rGoodStatistics[0]( CLK := stCycleDataNest1.LSS_Pass);
rBadStatistics[0]( CLK := stCycleDataNest1.LSS_Fail);
rGoodStatistics[1]( CLK := stCycleDataNest2.LSS_Pass);
rBadStatistics[1]( CLK := stCycleDataNest2.LSS_Fail);

IF 	rGoodStatistics[0].Q THEN
	
	stStatisticsHMI[4].nGood		:= stStatisticsHMI[4].nGood + 1;
	
END_IF
								
IF 	rBadStatistics[0].Q THEN
	
	stStatisticsHMI[4].nBad			:= stStatisticsHMI[4].nBad + 1;
	
END_IF

IF stStatisticsHMI[4].bResetGood THEN
	stStatisticsHMI[4].nGood		:= 0;
END_IF

IF stStatisticsHMI[4].bResetBad THEN
	stStatisticsHMI[4].nBad			:= 0;
END_IF

IF 	rGoodStatistics[1].Q THEN
	
	stStatisticsHMI[5].nGood		:= stStatisticsHMI[5].nGood + 1;
	
END_IF
								
IF 	rBadStatistics[1].Q THEN
	
	stStatisticsHMI[5].nBad			:= stStatisticsHMI[5].nBad + 1;
	
END_IF

IF stStatisticsHMI[5].bResetGood THEN
	stStatisticsHMI[5].nGood		:= 0;
END_IF

IF stStatisticsHMI[5].bResetBad THEN
	stStatisticsHMI[5].nBad			:= 0;
END_IF

IF (( stStatisticsHMI[4].nGood + stStatisticsHMI[4].nBad) <> 0) THEN
	
	rEfficency[0]							:= LREAL_TO_FMTSTR(in := (DINT_TO_REAL(stStatisticsHMI[4].nGood) /( DINT_TO_REAL(stStatisticsHMI[4].nGood) + DINT_TO_REAL(stStatisticsHMI[4].nBad))) * 100.0,iPrecision := 2, bRound := TRUE);
	stStatisticsHMI[4].nEfficency		:= CONCAT(STR1 := '%', STR2 := (rEfficency[0]));

ELSE stStatisticsHMI[4].nEfficency		:= CONCAT(STR1 := '%', STR2 := (DINT_TO_STRING(0)));
	
END_IF

IF (( stStatisticsHMI[5].nGood + stStatisticsHMI[5].nBad) <> 0) THEN
	
	rEfficency[1]							:= LREAL_TO_FMTSTR(in := (DINT_TO_REAL(stStatisticsHMI[5].nGood) /( DINT_TO_REAL(stStatisticsHMI[5].nGood) + DINT_TO_REAL(stStatisticsHMI[5].nBad))) * 100.0,iPrecision := 2, bRound := TRUE);
	stStatisticsHMI[5].nEfficency		:= CONCAT(STR1 := '%', STR2 := (rEfficency[1]));

ELSE stStatisticsHMI[5].nEfficency		:= CONCAT(STR1 := '%', STR2 := (DINT_TO_STRING(0)));
	
END_IF
END_ACTION

ACTION d_ACT_Set_Events_Station_3:
//IMMEDIATE FAULTS

stStationEvents[2].aEvents[0].bFault						:= TRUE;
stStationEvents[2].aEvents[0].bEventFlag					:= bError;
stStationEvents[2].aEvents[0].bEventText					:= 'Error Laser Snapshot';
stStationEvents[2].aEvents[0].sSolution						:= 'Check Laser Snapshot';


stStationEvents[2].aEvents[4].bFault						:= TRUE;
stStationEvents[2].aEvents[4].bEventTimer(IN := stLSS.Status.bBusy, PT := stTimers.tStation2TimeOut);
stStationEvents[2].aEvents[4].bEventFlag					:= stStationEvents[3].aEvents[4].bEventTimer.Q;
stStationEvents[2].aEvents[4].bEventText					:= 'Laser Snapshot Cycle Timeout';
stStationEvents[2].aEvents[4].sSolution						:= 'Reset Sytem';


//CYCLE STOP FAULT

stStationEvents[2].aEvents[24].bCycleStopRequest			:= TRUE;
stStationEvents[2].aEvents[24].bEventFlag					:= NOT bRun;
stStationEvents[2].aEvents[24].bEventText					:= 'Laser Snapshot is not in Run mode';
stStationEvents[2].aEvents[24].sSolution					:= 'Go to software and activate Run';
END_ACTION

ACTION e_ACT_HeightScalation:

//NEST LH
bScaledHeight1[1] := LSS_IO.nLH_HeightMeasurement_1-Offsets[1];
bScaledHeight1[2] := LSS_IO.nLH_HeightMeasurement_2-Offsets[2];
bScaledHeight1[3] := LSS_IO.nLH_HeightMeasurement_3-Offsets[3];
bScaledHeight1[4] := LSS_IO.nLH_HeightMeasurement_4-Offsets[4];
//NEST RH
bScaledHeight2[1] := LSS_IO.nRH_HeightMeasurement_1-Offsets[5];
bScaledHeight2[2] := LSS_IO.nRH_HeightMeasurement_2-Offsets[6];
bScaledHeight2[3] := LSS_IO.nRH_HeightMeasurement_3-Offsets[7];
bScaledHeight2[4] := LSS_IO.nRH_HeightMeasurement_4-Offsets[8];
END_ACTION

ACTION f_ACT_Measurement:

///////////////////////////////////////////////NEST 1//////////////////////////////////////////////
nHighLimit								:= nHeightSetPoint + nHeightTolerance;
nLowLimit								:= nHeightSetPoint - nHeightTolerance;
	

IF stLSS.CMD.LSS_CMD.Measurement1 THEN
	
IF 	(bScaledHeight1[1] < nHighLimit) AND
	(bScaledHeight1[1] > nLowLimit) THEN
									
	stCycleDataNest1.LSS_HeightPass[1]	:= TRUE;
	stCycleDataNest1.LSS_HeightFail[1]	:= FALSE;
									
ELSE
									
	stCycleDataNest1.LSS_HeightPass[1]	:= FALSE;
	stCycleDataNest1.LSS_HeightFail[1]	:= TRUE;
									
END_IF

IF 	(bScaledHeight1[2] < nHighLimit) AND
	(bScaledHeight1[2] > nLowLimit) THEN
									
	stCycleDataNest1.LSS_HeightPass[2]	:= TRUE;
	stCycleDataNest1.LSS_HeightFail[2]	:= FALSE;
									
ELSE
									
	stCycleDataNest1.LSS_HeightPass[2]	:= FALSE;
	stCycleDataNest1.LSS_HeightFail[2]	:= TRUE;
									
END_IF

IF 	(bScaledHeight1[3] < nHighLimit) AND
	(bScaledHeight1[3] > nLowLimit) THEN
									
	stCycleDataNest1.LSS_HeightPass[3]	:= TRUE;
	stCycleDataNest1.LSS_HeightFail[3]	:= FALSE;
									
ELSE
									
	stCycleDataNest1.LSS_HeightPass[3]	:= FALSE;
	stCycleDataNest1.LSS_HeightFail[3]	:= TRUE;
									
END_IF

IF 	(bScaledHeight1[4] < nHighLimit) AND
	(bScaledHeight1[4] > nLowLimit) THEN
									
	stCycleDataNest1.LSS_HeightPass[4]	:= TRUE;
	stCycleDataNest1.LSS_HeightFail[4]	:= FALSE;
									
ELSE
									
	stCycleDataNest1.LSS_HeightPass[4]	:= FALSE;
	stCycleDataNest1.LSS_HeightFail[4]	:= TRUE;
									
END_IF

IF stCycleDataNest1.LSS_HeightPass[1] AND stCycleDataNest1.LSS_HeightPass[2] AND
	stCycleDataNest1.LSS_HeightPass[3] AND stCycleDataNest1.LSS_HeightPass[4] THEN
	
	stCycleDataNest1.LSS_Pass			:= TRUE;
	stCycleDataNest1.LSS_Fail			:= FALSE;
	
ELSE 
	
	stCycleDataNest1.LSS_Pass			:= FALSE;
	stCycleDataNest1.LSS_Fail			:= TRUE;
	
END_IF

END_IF

///////////////////////////////////////////////NEST 2//////////////////////////////////////////////

IF stLSS.CMD.LSS_CMD.Measurement2 THEN
	
IF 	(bScaledHeight2[1] < nHighLimit) AND
	(bScaledHeight2[1] > nLowLimit) THEN
									
	stCycleDataNest2.LSS_HeightPass[1]	:= TRUE;
	stCycleDataNest2.LSS_HeightFail[1]	:= FALSE;
									
ELSE
									
	stCycleDataNest2.LSS_HeightPass[1]	:= FALSE;
	stCycleDataNest2.LSS_HeightFail[1]	:= TRUE;
									
END_IF

IF 	(bScaledHeight2[2] < nHighLimit) AND
	(bScaledHeight2[2] > nLowLimit) THEN
									
	stCycleDataNest2.LSS_HeightPass[2]	:= TRUE;
	stCycleDataNest2.LSS_HeightFail[2]	:= FALSE;
									
ELSE
									
	stCycleDataNest2.LSS_HeightPass[2]	:= FALSE;
	stCycleDataNest2.LSS_HeightFail[2]	:= TRUE;
									
END_IF

IF 	(bScaledHeight2[3] < nHighLimit) AND
	(bScaledHeight2[3] > nLowLimit) THEN
									
	stCycleDataNest2.LSS_HeightPass[3]	:= TRUE;
	stCycleDataNest2.LSS_HeightFail[3]	:= FALSE;
									
ELSE
									
	stCycleDataNest2.LSS_HeightPass[3]	:= FALSE;
	stCycleDataNest2.LSS_HeightFail[3]	:= TRUE;
									
END_IF

IF 	(bScaledHeight2[4] < nHighLimit) AND
	(bScaledHeight2[4] > nLowLimit) THEN
									
	stCycleDataNest2.LSS_HeightPass[4]	:= TRUE;
	stCycleDataNest2.LSS_HeightFail[4]	:= FALSE;
									
ELSE
									
	stCycleDataNest2.LSS_HeightPass[4]	:= FALSE;
	stCycleDataNest2.LSS_HeightFail[4]	:= TRUE;
									
END_IF

IF stCycleDataNest2.LSS_HeightPass[1] AND stCycleDataNest2.LSS_HeightPass[2] AND
	stCycleDataNest2.LSS_HeightPass[3] AND stCycleDataNest2.LSS_HeightPass[4] THEN
	
	stCycleDataNest2.LSS_Pass			:= TRUE;
	stCycleDataNest2.LSS_Fail			:= FALSE;
	
ELSE 
	
	stCycleDataNest2.LSS_Pass			:= FALSE;
	stCycleDataNest2.LSS_Fail			:= TRUE;
	
END_IF

END_IF
END_ACTION

ACTION g_ACT_Calibration:
tonCalibrationTrigger( IN := (bSetCalibrationHeight1 OR bSetCalibrationHeight2) AND (bResultsReady AND NOT bBusy), PT := T#500MS);

IF bSetCalibrationHeight1 THEN
	
	bTrigger										:= TRUE;
			
	CalibrationHeight1[1]						:= LSS_IO.nLH_HeightMeasurement_1;	
	CalibrationHeight1[2]						:= LSS_IO.nLH_HeightMeasurement_2;
	CalibrationHeight1[3]						:= LSS_IO.nLH_HeightMeasurement_3;
	CalibrationHeight1[4]						:= LSS_IO.nLH_HeightMeasurement_4;	

END_IF

IF bSetCalibrationHeight2 THEN
	
	bTrigger										:= TRUE;

	CalibrationHeight2[1]						:= LSS_IO.nRH_HeightMeasurement_1;	
	CalibrationHeight2[2]						:= LSS_IO.nRH_HeightMeasurement_2;
	CalibrationHeight2[3]						:= LSS_IO.nRH_HeightMeasurement_3;
	CalibrationHeight2[4]						:= LSS_IO.nRH_HeightMeasurement_4;

END_IF

IF tonCalibrationTrigger.Q THEN
	
	bSetCalibrationHeight1						:= FALSE;
	bSetCalibrationHeight2						:= FALSE;
	bResultsAcknowledge							:= TRUE;
	bTrigger									:= FALSE;
	

END_IF

tonResultAcknowledge(IN := NOT bSetCalibrationHeight1 AND NOT bSetCalibrationHeight2, PT := T#500MS);
rResultAcknowledge(CLK := tonResultAcknowledge.Q);

IF rResultAcknowledge.Q THEN
	
	bResultsAcknowledge							:= FALSE;

END_IF

Offsets[1]					:= CalibrationHeight1[1] - nHeightSetByCalibration;
Offsets[2]					:= CalibrationHeight1[2] - nHeightSetByCalibration;
Offsets[3]					:= CalibrationHeight1[3] - nHeightSetByCalibration;
Offsets[4]					:= CalibrationHeight1[4] - nHeightSetByCalibration;

Offsets[5]					:= CalibrationHeight2[1] - nHeightSetByCalibration;
Offsets[6]					:= CalibrationHeight2[2] - nHeightSetByCalibration;
Offsets[7]					:= CalibrationHeight2[3] - nHeightSetByCalibration;
Offsets[8]					:= CalibrationHeight2[4] - nHeightSetByCalibration;
END_ACTION

END_PROGRAM

// ---- POUs/B_STATIONS/B_3_CAMERA/B_3_1_PRG_Master_Camera.TcPOU
PROGRAM B_3_1_PRG_Master_Camera

VAR
	
	rGoodStatistics						: ARRAY [0..1] OF R_TRIG;
	rBadStatistics						: ARRAY [0..1] OF R_TRIG;
	rEfficency							: ARRAY [0..1] OF STRING(510);
	bEventsFlag							: ARRAY [0..100] OF BOOL;
/////////////////////////////////////////////////////////////////////////////////////I O/////////////////////////////////////////////////////////////////////////////////////	
	bError								: ARRAY [1..2] OF BOOL;
	rReset								: R_TRIG;
	bReset								: BOOL;
	bReady								: BOOL;
	bDone								: ARRAY [1..2] OF BOOL;
	bFail								: ARRAY [1..2] OF BOOL;
	bTrigger							: ARRAY [1..2] OF BOOL;
	bTriggerFail						: ARRAY [1..2] OF BOOL;
	bBusy								: ARRAY [1..2] OF BOOL;
	bGeneralBusy						: BOOL;
	bClearBuffer						: BOOL;
	tonTakingPicture					: TON;
	
	abReTakingPicture					: ARRAY [1..2] OF BOOL;

	
END_VAR

d_ACT_Set_Events_Station_3();
a_ACT_Ctrl_Station_3();
b_ACT_IO();
c_ACT_Statistics_Station_3();

ACTION a_ACT_Ctrl_Station_3:
/////////////////////////////////////////////////////////////////////////////////////UTILITIES/////////////////////////////////////////////////////////////////////////////////////
tonTakingPicture(IN := stCamera.State = E_Camera_State.TAKING_PICTURE_PART_PRESENT_INSPECTION OR
						stCamera.State = E_Camera_State.TAKING_PICTURE_CONTINUOUS_PART_PRESENT, PT := T#500MS);

/////////////////////////////////////////////////////////////////////////////////////CONDITIONS/////////////////////////////////////////////////////////////////////////////////////

IF bError[1] OR bError[2] OR stCamera.CMD.bAbort THEN
	
	stCamera.State						:= E_Camera_State.RESET_CMD;

END_IF

CASE stCamera.State OF
	
	E_Camera_State.ABORTED:
	
								
								
	
								IF  stCamera.CMD.bEnable THEN
									
									stCamera.State						:= E_Camera_State.HOMING;
								
								END_IF
													
	E_Camera_State.HOMING:
	
								IF bReady THEN
									
									stCamera.State						:= E_Camera_State.READY;
									
								END_IF
	
						
	E_Camera_State.READY:
								bClearBuffer							:= TRUE;
							
								IF stCamera.CMD.bExecute THEN
									
									IF stCamera.CMD.CameraCMD.PartPresent1 OR stCamera.CMD.CameraCMD.PartPresent2 THEN
										
										stCamera.State					:=	E_Camera_State.TAKING_PICTURE_PART_PRESENT_INSPECTION;
										
									ELSIF stCamera.CMD.CameraCMD.ContinuousPartPresent1 OR stCamera.CMD.CameraCMD.ContinuousPartPresent2 THEN
										
										stCamera.State					:=	E_Camera_State.TAKING_PICTURE_CONTINUOUS_PART_PRESENT;
										
									END_IF
									
								END_IF
	
	E_Camera_State.TAKING_PICTURE_PART_PRESENT_INSPECTION:
								
								bClearBuffer							:= FALSE;
								
								bTrigger[1]								:= stCamera.CMD.CameraCMD.PartPresent1;
								bTrigger[2]								:= stCamera.CMD.CameraCMD.PartPresent2;
								
								IF tonTakingPicture.Q THEN
									
									bTrigger[1]							:= FALSE;
									bTrigger[2]							:= FALSE;
								
									bPartPresentNest1 					:= Camera1_IO.bPartPresentResult;
									bPartPresentNest2 					:= Camera2_IO.bPartPresentResult;
								
									stCamera.State 						:= E_Camera_State.RESULTS;
																	
								END_IF
	
	E_Camera_State.TAKING_PICTURE_CONTINUOUS_PART_PRESENT:
	
								IF stPuls.bFlash2Hz THEN
									
									bTrigger[1] 						:= stCamera.CMD.CameraCMD.ContinuousPartPresent1;
									bTrigger[2] 						:= stCamera.CMD.CameraCMD.ContinuousPartPresent2;
									
								ELSE 
									
									bTrigger[1]							:= FALSE;
									bTrigger[2]							:= FALSE;
									
								END_IF
								
								IF tonTakingPicture.Q THEN
								
									bPartPresentNest1 					:= Camera1_IO.bPartPresentResult;
									bPartPresentNest2 					:= Camera2_IO.bPartPresentResult;
									
								END_IF
								
								IF NOT stCamera.CMD.CameraCMD.ContinuousPartPresent1 AND NOT stCamera.CMD.CameraCMD.ContinuousPartPresent2 THEN
									
									stCamera.State						:= E_Camera_State.RESET_CMD;
									
								END_IF

		E_Camera_State.RESULTS:		
			
								bTrigger[1]								:= FALSE;
								bTrigger[2]								:= FALSE;	
								
								IF (bPartPresentNest1 OR NOT stCamera.CMD.CameraCMD.PartPresent1) AND 
									(bPartPresentNest2 OR NOT stCamera.CMD.CameraCMD.PartPresent2) THEN
									
									stCycleDataNest1.Camera_Pass			:= Camera1_IO.bSeptumPositionResult;
									stCycleDataNest1.Camera_Fail			:= NOT Camera1_IO.bSeptumPositionResult;
									stCycleDataNest2.Camera_Pass			:= Camera2_IO.bSeptumPositionResult;
									stCycleDataNest2.Camera_Fail			:= NOT Camera2_IO.bSeptumPositionResult;
									
									
								END_IF
									
								
								stCamera.State							:= E_Camera_State.DONE;
								
		E_Camera_State.DONE:		
	
								IF stCamera.CMD.bAcknowledge THEN
									
									stCamera.CMD.bAcknowledge			:= FALSE;
									stCamera.State						:= E_Camera_State.RESET_CMD;
								
								END_IF
								
	E_Camera_State.RESET_CMD:						
	
								
									
								bTrigger[1]								:= FALSE;
								bTrigger[2]								:= FALSE;								
									
								IF  stCamera.CMD.bAbort THEN

									stCamera.State						:= E_Camera_State.ABORTED;
								
								ELSE 
									stCamera.State						:= E_Camera_State.READY;
								END_IF
									

ELSE stCamera.State						:= E_Camera_State.READY;
	
END_CASE
/////////////////////////////////////////////////////////////////////////////////////STATUS/////////////////////////////////////////////////////////////////////////////////////

stCamera.Status.bBusy		:= 	(stCamera.State	= E_Camera_State.TAKING_PICTURE_PART_PRESENT_INSPECTION) OR 
								(stCamera.State	= E_Camera_State.TAKING_PICTURE_CONTINUOUS_PART_PRESENT);
								
stCamera.Status.bDone		:=	stCamera.State	= E_Camera_State.DONE;
											
stCamera.Status.bError		:= 	stCamera.State	= E_Camera_State.ERROR;

stCamera.Status.bReady		:= 	stCamera.State	= E_Camera_State.READY;

stCamera.Status.bStopped	:= 	NOT stCamera.Status.bBusy;
END_ACTION

ACTION b_ACT_IO:


bError[1]								:= Camera1_IO.bError;
bError[2]								:= Camera2_IO.bError;

	
bReady									:=  (Camera1_IO.bReady AND Camera1_IO.bRun) AND (Camera2_IO.bReady AND Camera2_IO.bRun);
	
bDone[1]								:= Camera1_IO.bResultReady;
bDone[2]								:= Camera2_IO.bResultReady;
	
bGeneralBusy						:= bBusy[1] OR bBusy[2];



bBusy[1]								:= Camera1_IO.bBusy;
bBusy[2]								:= Camera2_IO.bBusy;

bTriggerFail[1]							:= Camera1_IO.bTriggerFail;
bTriggerFail[2]							:= Camera2_IO.bTriggerFail;

Camera1_IO.bReset						:= bReset;
Camera2_IO.bReset						:= bReset;

Camera1_IO.bTrigger						:= bTrigger[1] OR bCameraTrigger[1];	
Camera2_IO.bTrigger						:= bTrigger[2] OR bCameraTrigger[2];

IF bClearBuffer	THEN
	
	Camera1_IO.bClearBuffer				:= TRUE;
	Camera2_IO.bClearBuffer				:= TRUE;

ELSE

	Camera1_IO.bClearBuffer				:= FALSE;
	Camera2_IO.bClearBuffer				:= FALSE;

END_IF
	

//////////////////////////////////////////////////////////////////////HMI//////////////////////////////////////////////////////////////////////////////
bCameraSettingNo[1]						:= 2;
bCameraSettingNo[2]						:= 2;



Camera1_IO.bResetStatistics				:= bCameraResetStatistics[1];
Camera1_IO.bSettingNo					:= bCameraSettingNo[1];
Camera1_IO.bSettingVal					:= bCameraSettingVal[1];
Camera1_IO.bSetTreshold					:= bCameraSetTreshold[1];

Camera2_IO.bResetStatistics				:= bCameraResetStatistics[2];
Camera2_IO.bSettingNo					:= bCameraSettingNo[2];
Camera2_IO.bSettingVal					:= bCameraSettingVal[2];
Camera2_IO.bSetTreshold					:= bCameraSetTreshold[2];


//Camera1_IO.bTriggerFail

rReset( CLK := stCamera.CMD.bReset, Q => bReset);
END_ACTION

ACTION c_ACT_Statistics_Station_3:
stStatisticsHMI[6].sName			:= 'Vision System 1';
stStatisticsHMI[7].sName			:= 'Vision System 2';


rGoodStatistics[0]( CLK := stCycleDataNest1.Camera_Pass);
rBadStatistics[0]( CLK := stCycleDataNest1.Camera_Fail);
rGoodStatistics[1]( CLK := stCycleDataNest2.Camera_Pass);
rBadStatistics[1]( CLK := stCycleDataNest2.Camera_Fail);

IF 	rGoodStatistics[0].Q THEN
	
	stStatisticsHMI[6].nGood		:= stStatisticsHMI[6].nGood + 1;
	
END_IF
								
IF 	rBadStatistics[0].Q THEN
	
	stStatisticsHMI[6].nBad			:= stStatisticsHMI[6].nBad + 1;
	
END_IF

IF stStatisticsHMI[6].bResetGood THEN
	stStatisticsHMI[6].nGood		:= 0;
END_IF

IF stStatisticsHMI[6].bResetBad THEN
	stStatisticsHMI[6].nBad			:= 0;
END_IF

IF 	rGoodStatistics[1].Q THEN
	
	stStatisticsHMI[7].nGood		:= stStatisticsHMI[7].nGood + 1;
	
END_IF
								
IF 	rBadStatistics[1].Q THEN
	
	stStatisticsHMI[7].nBad			:= stStatisticsHMI[7].nBad + 1;
	
END_IF

IF stStatisticsHMI[7].bResetGood THEN
	stStatisticsHMI[7].nGood		:= 0;
END_IF

IF stStatisticsHMI[7].bResetBad THEN
	stStatisticsHMI[7].nBad			:= 0;
END_IF

IF (( stStatisticsHMI[6].nGood + stStatisticsHMI[6].nBad) <> 0) THEN
	
	rEfficency[0]							:= LREAL_TO_FMTSTR(in := (DINT_TO_REAL(stStatisticsHMI[6].nGood) /( DINT_TO_REAL(stStatisticsHMI[6].nGood) + DINT_TO_REAL(stStatisticsHMI[6].nBad))) * 100.0,iPrecision := 2, bRound := TRUE);
	stStatisticsHMI[6].nEfficency		:= CONCAT(STR1 := '%', STR2 := (rEfficency[0]));

ELSE stStatisticsHMI[6].nEfficency		:= CONCAT(STR1 := '%', STR2 := (DINT_TO_STRING(0)));
	
END_IF

IF (( stStatisticsHMI[7].nGood + stStatisticsHMI[7].nBad) <> 0) THEN
	
	rEfficency[1]							:= LREAL_TO_FMTSTR(in := (DINT_TO_REAL(stStatisticsHMI[7].nGood) /( DINT_TO_REAL(stStatisticsHMI[7].nGood) + DINT_TO_REAL(stStatisticsHMI[7].nBad))) * 100.0,iPrecision := 2, bRound := TRUE);
	stStatisticsHMI[7].nEfficency		:= CONCAT(STR1 := '%', STR2 := (rEfficency[1]));

ELSE stStatisticsHMI[7].nEfficency		:= CONCAT(STR1 := '%', STR2 := (DINT_TO_STRING(0)));
	
END_IF
END_ACTION

ACTION d_ACT_Set_Events_Station_3:
//IMMEDIATE FAULTS

stStationEvents[3].aEvents[0].bFault						:= TRUE;
stStationEvents[3].aEvents[0].bEventFlag					:= bError[1];
stStationEvents[3].aEvents[0].bEventText					:= 'Error camera 1';
stStationEvents[3].aEvents[0].sSolution						:= 'Check camera 1';

stStationEvents[3].aEvents[1].bFault						:= TRUE;
stStationEvents[3].aEvents[1].bEventFlag					:= bError[2];
stStationEvents[3].aEvents[1].bEventText					:= 'Error camera 2';
stStationEvents[3].aEvents[1].sSolution						:= 'Check camera 2';

stStationEvents[3].aEvents[4].bFault						:= TRUE;
stStationEvents[3].aEvents[4].bEventTimer(IN := stCamera.Status.bBusy, PT := stTimers.tStation3TimeOut);
stStationEvents[3].aEvents[4].bEventFlag					:= stStationEvents[3].aEvents[4].bEventTimer.Q;
stStationEvents[3].aEvents[4].bEventText					:= 'Camera Cycle Timeout';
stStationEvents[3].aEvents[4].sSolution						:= 'Reset Sytem';


//CYCLE STOP FAULT

stStationEvents[3].aEvents[20].bCycleStopRequest			:= TRUE;
stStationEvents[3].aEvents[20].bEventFlag					:= bTriggerFail[1];
stStationEvents[3].aEvents[20].bEventText					:= 'Trigger failed in camera 1';
stStationEvents[3].aEvents[20].sSolution					:= 'Check camera 1';

stStationEvents[3].aEvents[21].bCycleStopRequest			:= TRUE;
stStationEvents[3].aEvents[21].bEventFlag					:= bTriggerFail[2];
stStationEvents[3].aEvents[21].bEventText					:= 'Trigger failed in camera 2';
stStationEvents[3].aEvents[21].sSolution					:= 'Check camera 2';

stStationEvents[3].aEvents[24].bCycleStopRequest			:= TRUE;
stStationEvents[3].aEvents[24].bEventFlag					:= NOT Camera1_IO.bRun;
stStationEvents[3].aEvents[24].bEventText					:= 'Camera 1 is not in Run mode';
stStationEvents[3].aEvents[24].sSolution					:= 'Go to software and activate Run';

stStationEvents[3].aEvents[25].bCycleStopRequest			:= TRUE;
stStationEvents[3].aEvents[25].bEventFlag					:= NOT Camera2_IO.bRun;
stStationEvents[3].aEvents[25].bEventText					:= 'Camera 2 is not in Run mode';
stStationEvents[3].aEvents[25].sSolution					:= 'Go to software and activate Run';
END_ACTION

END_PROGRAM

// ---- POUs/B_STATIONS/B_1_LEAK_TEST/B_1_1_PRG_Master_Leak_Test.TcPOU
PROGRAM B_1_1_PRG_Master_Leak_Test

VAR

	tonStationStopped					: TON;
	tonExecute							: TON;
	rGoodStatistics						: ARRAY [0..1] OF R_TRIG;
	rBadStatistics						: ARRAY [0..1] OF R_TRIG;
	rEfficency							: ARRAY [0..1] OF STRING(510);
	
	tonWaitResults						: TON;
/////////////////////////////////////////////////////////////////////////////////////I O/////////////////////////////////////////////////////////////////////////////////////	

	bStopped							: ARRAY [0..1] OF BOOL;
	bError								: ARRAY [0..1] OF BOOL;
	bReady								: ARRAY [0..1] OF BOOL;
	bDone								: ARRAY [0..1] OF BOOL;
	bReset								: ARRAY [0..1] OF BOOL;
	bStart								: ARRAY [0..1] OF BOOL;
	bStop								: ARRAY [0..1] OF BOOL;	
	bBusy								: ARRAY [0..1] OF BOOL;	
	fLeakTestDone						: ARRAY [0..1] OF F_TRIG;	
	bLeakTestDone						: ARRAY [0..1] OF BOOL;	
	rPass								: ARRAY [0..1] OF R_TRIG;	
	bPass								: ARRAY [0..1] OF BOOL;	
	rFail								: ARRAY [0..1] OF R_TRIG;	
	bFail								: ARRAY [0..1] OF BOOL;
	rReset								: ARRAY [0..1] OF R_TRIG;

	
END_VAR

a_ACT_Ctrl_Station_1();
b_ACT_IO();
c_ACT_Statistics_Station_1();
d_ACT_Set_Events_Station_1();

ACTION a_ACT_Ctrl_Station_1:
/////////////////////////////////////////////////////////////////////////////////////UTILITIES/////////////////////////////////////////////////////////////////////////////////////
tonStationStopped( IN := bStopped[0] AND bStopped[1], PT := T#1S);
tonExecute(IN := stLeakTesters.State = E_LeakTester_State.RUN_LEAK_TESTERS, PT := T#500MS);
tonWaitResults(IN := (stLeakTesters.State = E_LeakTester_State.WAIT_RESULTS), PT := T#100MS);

/////////////////////////////////////////////////////////////////////////////////////CONDITIONS/////////////////////////////////////////////////////////////////////////////////////

IF stLeakTesters.CMD.bAbort OR bError[0] OR bError[1] THEN
								
	stLeakTesters.State											:= E_LeakTester_State.RESET;
	

END_IF



CASE stLeakTesters.State OF
	
	E_LeakTester_State.ABORTED:
	
								IF stLeakTesters.CMD.bEnable AND NOT bError[0] THEN
									stLeakTesters.State			:= E_LeakTester_State.HOMING;
								ELSIF bError[0] OR bError[1] THEN
									stLeakTesters.State			:= E_LeakTester_State.ERROR;
								END_IF
	
	E_LeakTester_State.HOMING:
	
								IF bReady[0] AND bReady[1] AND bStopped[0] AND bStopped[1] THEN
									stLeakTesters.State			:= E_LeakTester_State.READY;
								
								END_IF
								
	E_LeakTester_State.READY:
	
								IF stLeakTesters.CMD.bExecute THEN
									
									stLeakTesters.State			:= E_LeakTester_State.RUN_LEAK_TESTERS;
								
								END_IF
		
								
	E_LeakTester_State.RUN_LEAK_TESTERS:	
								
								IF stLeakTesters.CMD.LeakTestersCMD.RunLeakTester1 AND stLeakTesters.CMD.LeakTestersCMD.RunLeakTester2 THEN
										
										bStart[0]				:= TRUE;
										bStart[1]				:= TRUE;
									
								ELSIF stLeakTesters.CMD.LeakTestersCMD.RunLeakTester1 AND NOT stLeakTesters.CMD.LeakTestersCMD.RunLeakTester2 THEN
										
										bStart[0]				:= TRUE;
									
								ELSIF NOT stLeakTesters.CMD.LeakTestersCMD.RunLeakTester1 AND stLeakTesters.CMD.LeakTestersCMD.RunLeakTester2 THEN
										
										bStart[1]				:= TRUE;
									
								END_IF
								
								IF tonExecute.Q THEN
									
									stLeakTesters.State			:= E_LeakTester_State.WAIT_LEAK_TESTERS;
								
								END_IF
	
	E_LeakTester_State.WAIT_LEAK_TESTERS:
	
								IF stLeakTesters.CMD.LeakTestersCMD.RunLeakTester1 AND stLeakTesters.CMD.LeakTestersCMD.RunLeakTester2 THEN
										
										IF bLeakTestDone[0] AND bLeakTestDone[1] THEN
											
											stLeakTesters.State	:= E_LeakTester_State.WAIT_RESULTS;
											
										END_IF
									
								ELSIF stLeakTesters.CMD.LeakTestersCMD.RunLeakTester1 AND NOT stLeakTesters.CMD.LeakTestersCMD.RunLeakTester2 THEN
										
										IF bLeakTestDone[0]  THEN
											
											stLeakTesters.State	:= E_LeakTester_State.WAIT_RESULTS;
											
										END_IF
									
								ELSIF NOT stLeakTesters.CMD.LeakTestersCMD.RunLeakTester1 AND stLeakTesters.CMD.LeakTestersCMD.RunLeakTester2 THEN
										
										IF bLeakTestDone[1]  THEN
											
											stLeakTesters.State	:= E_LeakTester_State.WAIT_RESULTS;
											
										END_IF
									
								END_IF
	
	E_LeakTester_State.WAIT_RESULTS:
	
								IF tonWaitResults.Q THEN
									
									stLeakTesters.State	:= E_LeakTester_State.RESULTS;
									
								END_IF


		
	E_LeakTester_State.RESULTS:
								
								IF stLeakTesters.CMD.LeakTestersCMD.RunLeakTester1 THEN
									
									IF bPass[0] THEN
									
										stCycleDataNest1.LeakTest_Pass := TRUE;
										stCycleDataNest1.LeakTest_Fail := FALSE;
										
										stLeakTesters.State	:= E_LeakTester_State.DONE;
								
									ELSIF bFail[0] THEN
									
										stCycleDataNest1.LeakTest_Fail := TRUE;
										stCycleDataNest1.LeakTest_Pass := FALSE;
								
										stLeakTesters.State	:= E_LeakTester_State.DONE;
										
								END_IF
									
								END_IF
								
								IF stLeakTesters.CMD.LeakTestersCMD.RunLeakTester2 THEN
									
									IF bPass[1] THEN
									
										stCycleDataNest2.LeakTest_Pass := TRUE;
										stCycleDataNest2.LeakTest_Fail	:= FALSE;
										
										stLeakTesters.State	:= E_LeakTester_State.DONE;
								
									ELSIF bFail[1] THEN
									
										stCycleDataNest2.LeakTest_Fail	:= TRUE;
										stCycleDataNest2.LeakTest_Pass := FALSE;
										
										stLeakTesters.State	:= E_LeakTester_State.DONE;
								
								END_IF
									
								END_IF
								
								
								
		E_LeakTester_State.DONE:
								IF  stLeakTesters.CMD.bAcknowledge THEN
									
									stLeakTesters.CMD.bAcknowledge := FALSE;
									stLeakTesters.State			:= E_LeakTester_State.RESET;
									
								END_IF	
								
								
								
	E_LeakTester_State.RESET:
	

								bStart[0]						:= FALSE;
								bStart[1]						:= FALSE;
								bReset[0]						:= FALSE;
								bReset[1]						:= FALSE;
								bStop[0]						:= FALSE;
								bStop[1]						:= FALSE;
								bLeakTestDone[0]				:= FALSE;
								bLeakTestDone[1]				:= FALSE;
								bPass[0]						:= FALSE;
								bPass[1]						:= FALSE;
								bFail[0]						:= FALSE;
								bFail[1]						:= FALSE;
								
								IF bError[0] OR bError[1] THEN

									stLeakTesters.State		:= E_LeakTester_State.ERROR;

								ELSIF stLeakTesters.CMD.bAbort OR stLeakTesters.CMD.bEndCycle THEN
									
									stLeakTesters.State			:= E_LeakTester_State.ABORTED;
									
								ELSE stLeakTesters.State			:= E_LeakTester_State.READY;
								
								END_IF
								
								
								
	E_LeakTester_State.STOPPING: 
	
								bStop[0]						:= TRUE;
								bStop[1]						:= TRUE;
								
								IF tonStationStopped.Q THEN
									
									stLeakTesters.State			:= E_LeakTester_State.RESET;
									
								END_IF
	
	E_LeakTester_State.ERROR:
	
								IF NOT bError[0] AND bError[1] THEN
									
									stLeakTesters.State						:= E_LeakTester_State.ABORTED;
									
								END_IF

ELSE stLeakTesters.State := E_LeakTester_State.ABORTED;
	
END_CASE
/////////////////////////////////////////////////////////////////////////////////////STATUS/////////////////////////////////////////////////////////////////////////////////////

stLeakTesters.Status.bBusy	:= 	stLeakTesters.State = E_LeakTester_State.STOPPING OR
								stLeakTesters.State = E_LeakTester_State.HOMING OR
								stLeakTesters.State = E_LeakTester_State.RUN_LEAK_TESTERS OR
								stLeakTesters.State = E_LeakTester_State.WAIT_LEAK_TESTERS;

stLeakTesters.Status.bDone	:= 	stLeakTesters.State = E_LeakTester_State.DONE;

stLeakTesters.Status.bError	:= 	stLeakTesters.State = E_LeakTester_State.ERROR;	

stLeakTesters.Status.bReady	:=	stLeakTesters.State = E_LeakTester_State.READY;

stLeakTesters.Status.bStopped := NOT stLeakTesters.Status.bBusy;
END_ACTION

ACTION b_ACT_IO:


bStopped[0]								:= NOT LeakTester1_IO.sti28General_I_O.bTestActiveLiveData;
bStopped[1]								:= NOT LeakTester2_IO.sti28General_I_O.bTestActiveLiveData;
bError[0]								:= LeakTester1_IO.sti28General_I_O.bMalfunction;
bError[1]								:= LeakTester2_IO.sti28General_I_O.bMalfunction;
bReady[0]								:= LeakTester1_IO.sti28General_I_O.bInstrumentReady;
bReady[1]								:= LeakTester2_IO.sti28General_I_O.bInstrumentReady;
LeakTester1_IO.sti28General_I_O.bReset	:= bReset[0] OR bLeaktester1_Reset;	
LeakTester2_IO.sti28General_I_O.bReset	:= bReset[1] OR bLeaktester2_Reset;	
LeakTester1_IO.sti28General_I_O.bStart	:= bStart[0] OR bLeaktester1_Start;
LeakTester2_IO.sti28General_I_O.bStart	:= bStart[1] OR bLeaktester2_Start;
LeakTester1_IO.sti28General_I_O.bStop	:= bStop[0] OR bLeaktester1_Stop OR stLeakTesters.CMD.bAbort;
LeakTester2_IO.sti28General_I_O.bStop	:= bStop[1] OR bLeaktester2_Stop OR stLeakTesters.CMD.bAbort;



rReset[0](CLK := stLeakTesters.CMD.bReset, Q => bReset[0]);
rReset[1](CLK := stLeakTesters.CMD.bReset, Q => bReset[1]);

fLeakTestDone[0](CLK := LeakTester1_IO.sti28General_I_O.bTestActiveLiveData);
fLeakTestDone[1](CLK := LeakTester2_IO.sti28General_I_O.bTestActiveLiveData);
rPass[0](CLK := LeakTester1_IO.sti28General_I_O.bProgramAccept);
rPass[1](CLK := LeakTester2_IO.sti28General_I_O.bProgramAccept);
rFail[0](CLK := LeakTester1_IO.sti28General_I_O.bProgramReject);
rFail[1](CLK := LeakTester2_IO.sti28General_I_O.bProgramReject);



IF fLeakTestDone[0].Q THEN
	
	bLeakTestDone[0]					:= TRUE;
	
END_IF

IF fLeakTestDone[1].Q THEN
	
	bLeakTestDone[1]					:= TRUE;
	
END_IF

IF rPass[0].Q THEN
	
	bPass[0]							:= TRUE;

END_IF

IF rPass[1].Q THEN
	
	bPass[1]							:= TRUE;

END_IF

IF rFail[0].Q THEN
	
	bFail[0]							:= TRUE;

END_IF

IF rFail[1].Q THEN
	
	bFail[1]							:= TRUE;

END_IF
END_ACTION

ACTION c_ACT_Statistics_Station_1:
stStatisticsHMI[2].sName			:= 'LEAK TESTER 1';
stStatisticsHMI[3].sName			:= 'LEAK TESTER 2';


rGoodStatistics[0]( CLK := stCycleDataNest1.LeakTest_Pass );
rGoodStatistics[1]( CLK := stCycleDataNest2.LeakTest_Pass );
rBadStatistics[0] ( CLK := stCycleDataNest1.LeakTest_Fail );
rBadStatistics[1] ( CLK := stCycleDataNest2.LeakTest_Fail );

IF 	rGoodStatistics[0].Q THEN
	
	stStatisticsHMI[2].nGood		:= stStatisticsHMI[2].nGood + 1;
	
END_IF
								
IF 	rBadStatistics[0].Q THEN
	
	stStatisticsHMI[2].nBad			:= stStatisticsHMI[2].nBad + 1;
	
END_IF

IF stStatisticsHMI[2].bResetGood THEN
	stStatisticsHMI[2].nGood		:= 0;
END_IF

IF stStatisticsHMI[2].bResetBad THEN
	stStatisticsHMI[2].nBad			:= 0;
END_IF


IF 	rGoodStatistics[1].Q THEN
	
	stStatisticsHMI[3].nGood		:= stStatisticsHMI[3].nGood + 1;
	
END_IF
								
IF 	rBadStatistics[1].Q THEN
	
	stStatisticsHMI[3].nBad			:= stStatisticsHMI[3].nBad + 1;
	
END_IF

IF stStatisticsHMI[3].bResetGood THEN
	stStatisticsHMI[3].nGood		:= 0;
END_IF

IF stStatisticsHMI[3].bResetBad THEN
	stStatisticsHMI[3].nBad			:= 0;
END_IF



IF (( stStatisticsHMI[2].nGood + stStatisticsHMI[2].nBad) <> 0) THEN
	
	rEfficency[0]							:= LREAL_TO_FMTSTR(in := (DINT_TO_REAL(stStatisticsHMI[2].nGood) /( DINT_TO_REAL(stStatisticsHMI[2].nGood) + DINT_TO_REAL(stStatisticsHMI[2].nBad))) * 100.0,iPrecision := 2, bRound := TRUE);
	stStatisticsHMI[2].nEfficency		:= CONCAT(STR1 := '%', STR2 := (rEfficency[0]));

ELSE stStatisticsHMI[2].nEfficency		:= CONCAT(STR1 := '%', STR2 := (DINT_TO_STRING(0)));
	
END_IF

IF (( stStatisticsHMI[3].nGood + stStatisticsHMI[3].nBad) <> 0) THEN
	
	rEfficency[1]							:= LREAL_TO_FMTSTR(in := (DINT_TO_REAL(stStatisticsHMI[3].nGood) /( DINT_TO_REAL(stStatisticsHMI[3].nGood) + DINT_TO_REAL(stStatisticsHMI[3].nBad))) * 100.0,iPrecision := 2, bRound := TRUE);
	stStatisticsHMI[3].nEfficency		:= CONCAT(STR1 := '%', STR2 := (rEfficency[1]));

ELSE stStatisticsHMI[3].nEfficency		:= CONCAT(STR1 := '%', STR2 := (DINT_TO_STRING(0)));
	
END_IF
END_ACTION

ACTION d_ACT_Set_Events_Station_1:
//IMMEDIATE FAULTS

stStationEvents[1].aEvents[0].bFault						:= TRUE;
stStationEvents[1].aEvents[0].bEventTimer( IN := (stLeakTesters.State = E_LeakTester_State.RUN_LEAK_TESTERS) OR (stLeakTesters.State = E_LeakTester_State.WAIT_LEAK_TESTERS), PT := stTimers.tStation1TimeOut);
stStationEvents[1].aEvents[0].bEventFlag					:= stStationEvents[1].aEvents[0].bEventTimer.Q;
stStationEvents[1].aEvents[0].bEventText					:= 'Leak tester cycle Timeout';
stStationEvents[1].aEvents[0].sSolution						:= 'Reset System';



//CYCLE STOP REQUEST

stStationEvents[1].aEvents[20].bCycleStopRequest				:= TRUE;
stStationEvents[1].aEvents[20].bEventFlag					:= NOT bReady[0] AND (stLeakTesters.State = E_LeakTester_State.HOMING);// AND (stLeakTesters.State = E_LeakTester_State.HOMING);
stStationEvents[1].aEvents[20].bEventText					:= 'Leak Tester 1 not ready';
stStationEvents[1].aEvents[20].sSolution						:= 'Check Leak tester 1';

stStationEvents[1].aEvents[21].bCycleStopRequest				:= TRUE;
stStationEvents[1].aEvents[21].bEventFlag					:= NOT bReady[1] AND (stLeakTesters.State = E_LeakTester_State.HOMING);// AND (stLeakTesters.State = E_LeakTester_State.HOMING);
stStationEvents[1].aEvents[21].bEventText					:= 'Leak Tester 2 not ready';
stStationEvents[1].aEvents[21].sSolution						:= 'Check Leak tester 2';

stStationEvents[1].aEvents[22].bCycleStopRequest			:= TRUE;
stStationEvents[1].aEvents[22].bEventFlag					:= bError[0] AND bNest1Flag;
stStationEvents[1].aEvents[22].bEventText					:= 'Leak Tester 1 malfunction';
stStationEvents[1].aEvents[22].sSolution					:= 'Check Leak tester 1';

stStationEvents[1].aEvents[23].bCycleStopRequest			:= TRUE;
stStationEvents[1].aEvents[23].bEventFlag					:=  bError[1] AND bNest2Flag;
stStationEvents[1].aEvents[23].bEventText					:= 'Leak Tester 2 malfunction';
stStationEvents[1].aEvents[23].sSolution					:= 'Check Leak tester 2';

stStationEvents[1].aEvents[24].bCycleStopRequest			:= TRUE;
stStationEvents[1].aEvents[24].rEventTrigger( CLK := LeakTester1_IO.sti28LasResult.inPartEvaluation = 13);
stStationEvents[1].aEvents[24].bEventFlag					:=  stStationEvents[1].aEvents[24].rEventTrigger.Q;
stStationEvents[1].aEvents[24].bEventText					:= 'Leak Tester 1 Low Pressure';
stStationEvents[1].aEvents[24].sSolution					:= 'Check Leak tester 1 pneumatic circuit ';

stStationEvents[1].aEvents[25].bCycleStopRequest			:= TRUE;
stStationEvents[1].aEvents[25].rEventTrigger( CLK := LeakTester1_IO.sti28LasResult.inPartEvaluation = 14);
stStationEvents[1].aEvents[25].bEventFlag					:=  stStationEvents[1].aEvents[25].rEventTrigger.Q;
stStationEvents[1].aEvents[25].bEventText					:= 'Leak Tester 1 High Pressure';
stStationEvents[1].aEvents[25].sSolution					:= 'Check Leak tester 1 parameters';

stStationEvents[1].aEvents[26].bCycleStopRequest			:= TRUE;
stStationEvents[1].aEvents[26].rEventTrigger( CLK := LeakTester2_IO.sti28LasResult.inPartEvaluation = 13);
stStationEvents[1].aEvents[26].bEventFlag					:=  stStationEvents[1].aEvents[26].rEventTrigger.Q;
stStationEvents[1].aEvents[26].bEventText					:= 'Leak Tester 2 Low Pressure';
stStationEvents[1].aEvents[26].sSolution					:= 'Check Leak tester 2 pneumatic circuit ';

stStationEvents[1].aEvents[27].bCycleStopRequest			:= TRUE;
stStationEvents[1].aEvents[27].rEventTrigger( CLK := LeakTester2_IO.sti28LasResult.inPartEvaluation = 14);
stStationEvents[1].aEvents[27].bEventFlag					:=  stStationEvents[1].aEvents[27].rEventTrigger.Q;
stStationEvents[1].aEvents[27].bEventText					:= 'Leak Tester 2 High Pressure';
stStationEvents[1].aEvents[27].sSolution					:= 'Check Leak tester 2 parameters';

//Message
(*
stStationEvents[1].aEvents[3].bMessage						:= TRUE;
stStationEvents[1].aEvents[3].bEventFlag					:= bEventsFlag[3];
stStationEvents[1].aEvents[3].bEventText					:= 'Message 3';
stStationEvents[1].aEvents[3].sSolution						:= '';*)
END_ACTION

END_PROGRAM

// ---- POUs/B_STATIONS/B_4_PROCESS_CYLINDER__SLIDE_DOOR_VACUUM_CYLINDER/B_4_1_PRG_Master_ProcessCylinder.TcPOU
PROGRAM B_4_1_PRG_Master_ProcessCylinder

VAR

	
	
/////////////////////////////////////////////////////////////////////////////////////I O/////////////////////////////////////////////////////////////////////////////////////	
	bExtended							: ARRAY[1..2] OF BOOL;
	bRetracted							: ARRAY[1..2] OF BOOL;
	bExtend								: ARRAY[1..2] OF BOOL;
	bRetract							: ARRAY[1..2] OF BOOL;
	
	bHoldPart							: ARRAY[1..2] OF BOOL;
	tonPartReleased						: ARRAY[1..2] OF TON;
	tonHoldPart							: ARRAY[1..2] OF TON;
	
	bProcessDoorClosed					: BOOL;
	
END_VAR

d_ACT_Set_Events_Station_4A();
a_ACT_Ctrl_Station_4A();
b_ACT_IO_A();

ACTION a_ACT_Ctrl_Station_4A:
/////////////////////////////////////////////////////////////////////////////////////UTILITIES/////////////////////////////////////////////////////////////////////////////////////

IF stProcessCylinder.CMD.bAbort THEN
	
	stProcessCylinder.State												:= E_ProcessCylinder_State.RESET;
	bHoldPart[1]														:= FALSE;
	bHoldPart[2]														:= FALSE;

END_IF

/////////////////////////////////////////////////////////////////////////////////////CONDITIONS/////////////////////////////////////////////////////////////////////////////////////

CASE stProcessCylinder.State OF
	
	E_ProcessCylinder_State.ABORTED:
	
								IF stProcessCylinder.CMD.bEnable THEN
									
									stProcessCylinder.State				:= E_ProcessCylinder_State.HOMING;
								
								END_IF
								
	E_ProcessCylinder_State.HOMING:
	
								bHoldPart[1]							:= FALSE;
								bHoldPart[2]							:= FALSE;
	
								IF NOT bRetracted[1] AND (NOT bHoldPart[1] AND bProcessDoorClosed) THEN
									
									bRetract[1]							:= TRUE;
									
								END_IF
								
								IF NOT bRetracted[2] AND (NOT bHoldPart[2] AND bProcessDoorClosed) THEN
									
									bRetract[2]							:= TRUE;
									
								END_IF
								
								
								IF bRetracted[1] AND bRetracted[2] THEN
									
									bRetract[1]							:= FALSE;
									bRetract[2]							:= FALSE;
									stProcessCylinder.State				:= E_ProcessCylinder_State.READY;
									
								
								END_IF
	
	E_ProcessCylinder_State.READY:
	
								IF stProcessCylinder.CMD.bExecute AND (stProcessCylinder.CMD.ProcessCylinderCMD.ExtendCylinder1 OR stProcessCylinder.CMD.ProcessCylinderCMD.ExtendCylinder2) THEN

									stProcessCylinder.State				:= E_ProcessCylinder_State.EXTEND;
									
								ELSIF stProcessCylinder.CMD.bExecute AND (stProcessCylinder.CMD.ProcessCylinderCMD.RetractCylinder1 OR stProcessCylinder.CMD.ProcessCylinderCMD.RetractCylinder2) THEN
									
									stProcessCylinder.State				:= E_ProcessCylinder_State.RETRACT;

								ELSIF stProcessCylinder.CMD.bExecute AND (stProcessCylinder.CMD.ProcessCylinderCMD.ExtendPartHolder1 OR stProcessCylinder.CMD.ProcessCylinderCMD.ExtendPartHolder2) THEN

									stProcessCylinder.State				:= E_ProcessCylinder_State.HOLD_PART;	

								ELSIF stProcessCylinder.CMD.bExecute AND (stProcessCylinder.CMD.ProcessCylinderCMD.RetractPartHolder1 OR stProcessCylinder.CMD.ProcessCylinderCMD.RetractPartHolder2) THEN

									stProcessCylinder.State				:= E_ProcessCylinder_State.RELEASE_PART;			
																		
								END_IF
	
	E_ProcessCylinder_State.EXTEND:
	
								bExtend[1]									:= stProcessCylinder.CMD.ProcessCylinderCMD.ExtendCylinder1;
								bExtend[2]									:= stProcessCylinder.CMD.ProcessCylinderCMD.ExtendCylinder2;
								
								IF (bExtended[1] OR NOT stProcessCylinder.CMD.ProcessCylinderCMD.ExtendCylinder1) AND (bExtended[2] OR NOT stProcessCylinder.CMD.ProcessCylinderCMD.ExtendCylinder2) THEN
									
									stProcessCylinder.State			:= E_ProcessCylinder_State.DONE;

								END_IF
								
	E_ProcessCylinder_State.RETRACT:
	
								bRetract[1]									:= stProcessCylinder.CMD.ProcessCylinderCMD.RetractCylinder1;
								bRetract[2]									:= stProcessCylinder.CMD.ProcessCylinderCMD.RetractCylinder2;
								
								
								IF (bRetracted[1] OR NOT stProcessCylinder.CMD.ProcessCylinderCMD.RetractCylinder1) AND (bRetracted[2] OR NOT stProcessCylinder.CMD.ProcessCylinderCMD.RetractCylinder2) THEN
									
									stProcessCylinder.State			:= E_ProcessCylinder_State.DONE;

								END_IF
								
	E_ProcessCylinder_State.HOLD_PART:
	
								bHoldPart[1]								:= stProcessCylinder.CMD.ProcessCylinderCMD.ExtendPartHolder1;
								bHoldPart[2]								:= stProcessCylinder.CMD.ProcessCylinderCMD.ExtendPartHolder2;
								
								
								IF (tonHoldPart[1].Q OR NOT stProcessCylinder.CMD.ProcessCylinderCMD.ExtendPartHolder1) AND (tonHoldPart[2].Q OR NOT stProcessCylinder.CMD.ProcessCylinderCMD.ExtendPartHolder2) THEN
									
									stProcessCylinder.State			:= E_ProcessCylinder_State.DONE;

								END_IF
								
	E_ProcessCylinder_State.RELEASE_PART:
	
								bHoldPart[1]								:= FALSE;
								bHoldPart[2]								:= FALSE;
								
								
								IF (tonPartReleased[1].Q OR NOT stProcessCylinder.CMD.ProcessCylinderCMD.RetractPartHolder1) AND (tonPartReleased[2].Q OR NOT stProcessCylinder.CMD.ProcessCylinderCMD.RetractPartHolder2) THEN
									
									stProcessCylinder.State			:= E_ProcessCylinder_State.DONE;

								END_IF
								
	E_ProcessCylinder_State.DONE:
	
								IF stProcessCylinder.CMD.bAcknowledge THEN
									
									stProcessCylinder.CMD.bAcknowledge		:= FALSE;
									stProcessCylinder.State					:= E_ProcessCylinder_State.RESET;
								
								END_IF
	
	
	E_ProcessCylinder_State.RESET:	
	
								bExtend[1]									:= FALSE;								
								bRetract[1]									:= FALSE;
								bExtend[2]									:= FALSE;								
								bRetract[2]									:= FALSE;
								
								IF NOT stProcessCylinder.CMD.bAbort AND NOT stProcessCylinder.CMD.bEndCycle THEN
									
									stProcessCylinder.State					:= E_ProcessCylinder_State.READY;
									
								ELSE stProcessCylinder.State					:= E_ProcessCylinder_State.ABORTED;
								END_IF
									

ELSE stProcessCylinder.State	:= E_ProcessCylinder_State.ABORTED;
	
END_CASE
/////////////////////////////////////////////////////////////////////////////////////STATUS/////////////////////////////////////////////////////////////////////////////////////

stProcessCylinder.Status.bBusy		:= 	stProcessCylinder.State	= E_ProcessCylinder_State.EXTEND OR
										stProcessCylinder.State	= E_ProcessCylinder_State.RETRACT OR 
										stProcessCylinder.State	= E_ProcessCylinder_State.RELEASE_PART OR 
										stProcessCylinder.State	= E_ProcessCylinder_State.HOLD_PART OR 
										stProcessCylinder.State	= E_ProcessCylinder_State.STOPPING;
								
stProcessCylinder.Status.bDone		:=	stProcessCylinder.State	= E_ProcessCylinder_State.DONE;

stProcessCylinder.Status.bReady		:= 	stProcessCylinder.State	= E_ProcessCylinder_State.READY;

stProcessCylinder.Status.bStopped	:= 	NOT stProcessCylinder.Status.bBusy;

stProcessCylinder.Status.bHomed		:= bRetracted[1] AND bRetracted[2];
END_ACTION

ACTION b_ACT_IO_A:

bExtended[1]								:= dw_T08_EL1809.iProcessCylinderExtended1;
bRetracted[1]								:= dw_T08_EL1809.iProcessCylinderRetracted1;
bExtended[2]								:= dw_T08_EL1809.iProcessCylinderExtended2;
bRetracted[2]								:= dw_T08_EL1809.iProcessCylinderRetracted2;

IF (bHoldPart[1] OR bHoldPart1) AND bExtended[1] THEN
	
	dw_T09_EL2809.qPartHolder1				:= TRUE;
	
ELSE

 dw_T09_EL2809.qPartHolder1				:= FALSE;

END_IF

IF (bHoldPart[2] OR bHoldPart2) AND bExtended[2] THEN
	
	dw_T10_EL2809.qPartHolder2				:= TRUE;
	
ELSE dw_T10_EL2809.qPartHolder2				:= FALSE;

END_IF

tonHoldPart[1](IN := NOT dw_T09_EL2809.qPartHolder1, PT := T#1S);
tonHoldPart[2](IN := NOT dw_T10_EL2809.qPartHolder2, PT := T#1S);

tonPartReleased[1](IN := NOT bHoldPart[1], PT := T#1S);
tonPartReleased[2](IN := NOT bHoldPart[2], PT := T#1S);

IF (bExtend[1] OR bProcessCtlinderExtend1) AND (tonPartReleased[1].Q AND bProcessDoorClosed) THEN
	
	dw_T09_EL2809.qExtendProcessCylinder1	:= TRUE ;
	dw_T09_EL2809.qRetractProcessCylinder1	:= FALSE;

ELSIF (bRetract[1] OR bProcessCtlinderRetract1) AND (tonPartReleased[1].Q AND bProcessDoorClosed )  THEN
	
	dw_T09_EL2809.qExtendProcessCylinder1	:= FALSE;
	dw_T09_EL2809.qRetractProcessCylinder1	:= TRUE;
	
ELSIF stMachineStatus.bFault THEN
	
	dw_T09_EL2809.qExtendProcessCylinder1	:= FALSE;
	dw_T09_EL2809.qRetractProcessCylinder1	:= FALSE;

END_IF

IF (bExtend[2] OR bProcessCtlinderExtend2) AND (tonPartReleased[2].Q AND bProcessDoorClosed) THEN
	
	dw_T10_EL2809.qExtendProcessCylinder2	:= TRUE ;
	dw_T10_EL2809.qRetractProcessCylinder2	:= FALSE;

ELSIF (bRetract[2] OR bProcessCtlinderRetract2) AND (tonPartReleased[2].Q AND bProcessDoorClosed)  THEN
	
	dw_T10_EL2809.qExtendProcessCylinder2	:= FALSE;
	dw_T10_EL2809.qRetractProcessCylinder2	:= TRUE;
	
ELSIF stMachineStatus.bFault THEN
	
	dw_T10_EL2809.qExtendProcessCylinder2	:= FALSE;
	dw_T10_EL2809.qRetractProcessCylinder2	:= FALSE;

END_IF


bProcessDoorClosed := dw_T05_EL1918.iProcessDoorClosed1 AND dw_T05_EL1918.iProcessDoorClosed2 AND dw_T05_EL1918.iProcessDoorFB;


bEnable_Holder[1]							:= bExtended[1];
bEnable_Holder[2]							:= bExtended[2];

bEnable_ProcessCylinder[1]					:= bProcessDoorClosed AND tonHoldPart[1].Q;
bEnable_ProcessCylinder[2]					:= bProcessDoorClosed AND tonHoldPart[2].Q;

bPartHeld[1]								:= bExtended[1] AND dw_T09_EL2809.qPartHolder1;
bPartHeld[2]								:= bExtended[2] AND dw_T10_EL2809.qPartHolder2;
END_ACTION

ACTION d_ACT_Set_Events_Station_4A:
//FAULTS 0..9

stStationEvents[4].aEvents[0].bEventTimer( IN := (bExtend[1] AND NOT bExtended[1]), PT := T#3S);
stStationEvents[4].aEvents[0].bFault						:= TRUE;
stStationEvents[4].aEvents[0].bEventFlag					:= stStationEvents[3].aEvents[0].bEventTimer.Q;
stStationEvents[4].aEvents[0].bEventText					:= 'Process Cylinder 1 extend timeout';
stStationEvents[4].aEvents[0].sSolution						:= 'Check cylinder, neumatic connections and sensors';

stStationEvents[4].aEvents[1].bEventTimer( IN := (bRetract[1] AND NOT bRetracted[1]), PT := T#3S);
stStationEvents[4].aEvents[1].bFault						:= TRUE;
stStationEvents[4].aEvents[1].bEventFlag					:= stStationEvents[3].aEvents[1].bEventTimer.Q;
stStationEvents[4].aEvents[1].bEventText					:= 'Process Cylinder retract timeout';
stStationEvents[4].aEvents[1].sSolution						:= 'Check cylinder, neumatic connections and sensors';

stStationEvents[4].aEvents[2].bEventTimer( IN := (bExtend[2] AND NOT bExtended[2]), PT := T#3S);
stStationEvents[4].aEvents[2].bFault						:= TRUE;
stStationEvents[4].aEvents[2].bEventFlag					:= stStationEvents[3].aEvents[2].bEventTimer.Q;
stStationEvents[4].aEvents[2].bEventText					:= 'Process Cylinder 2 extend timeout';
stStationEvents[4].aEvents[2].sSolution						:= 'Check cylinder, neumatic connections and sensors';

stStationEvents[4].aEvents[2].bEventTimer( IN := (bRetract[2] AND NOT bRetracted[2]), PT := T#3S);
stStationEvents[4].aEvents[2].bFault						:= TRUE;
stStationEvents[4].aEvents[2].bEventFlag					:= stStationEvents[3].aEvents[3].bEventTimer.Q;
stStationEvents[4].aEvents[2].bEventText					:= 'Process Cylinder retract timeout';
stStationEvents[4].aEvents[2].sSolution						:= 'Check cylinder, neumatic connections and sensors';


//CYCLE STOP REQUEST 30..39

(*stStationEvents[3].aEvents[2].bCycleStopRequest			:= TRUE;
stStationEvents[3].aEvents[2].bEventFlag					:= ;
stStationEvents[3].aEvents[2].bEventText					:= 'ST1 EVENT 7';*)
END_ACTION

END_PROGRAM

// ---- POUs/B_STATIONS/B_4_PROCESS_CYLINDER__SLIDE_DOOR_VACUUM_CYLINDER/B_4_2_PRG_Master_ProcessDoor.TcPOU
PROGRAM B_4_2_PRG_Master_ProcessDoor

VAR

	bEventsFlag							: ARRAY [0..100] OF BOOL;
/////////////////////////////////////////////////////////////////////////////////////I O/////////////////////////////////////////////////////////////////////////////////////	
	
	bOpenDoor							: BOOL;
	bCloseDoor							: BOOL;
	bCloseDoorHMI						: BOOL;
	bOpenDoorHMI						: BOOL;
	bDoorClosed							: BOOL;
	tonDoorOpened						: TON;
	bDoorOpened							: BOOL;	
	
END_VAR

d_ACT_Set_Events_Station_4B();
a_ACT_Ctrl_Station_4B();
b_ACT_IO_B();
c_Manual();

ACTION a_ACT_Ctrl_Station_4B:
/////////////////////////////////////////////////////////////////////////////////////UTILITIES/////////////////////////////////////////////////////////////////////////////////////

/////////////////////////////////////////////////////////////////////////////////////CONDITIONS/////////////////////////////////////////////////////////////////////////////////////
IF stProcessDoor.State <> E_ProcessDoor_State.HOMING THEN
	
	bDoorClosingInitFlag											:= FALSE;

END_IF


IF stProcessDoor.CMD.bAbort THEN
	
	stProcessDoor.State				:= E_ProcessDoor_State.RESET;
	
ELSIF stProcessDoor.CMD.bEndCycle THEN
	
	stProcessDoor.State				:= E_ProcessDoor_State.STOPPING;

END_IF

CASE stProcessDoor.State OF
	
	E_ProcessDoor_State.ABORTED:
	
								IF stProcessDoor.CMD.bEnable THEN
									
									stProcessDoor.State				:= E_ProcessDoor_State.HOMING;
								
								END_IF
								
		E_ProcessDoor_State.HOMING: 
		
								IF NOT stProcessCylinder.Status.bHomed OR NOT stVacuumCylinder.Status.bHomed THEN
									
									bCloseDoor						:= TRUE;
									bOpenDoor						:= FALSE;
									
									IF NOT bDoorClosed AND bCloseDoor THEN
										
										bDoorClosingInitFlag		:= TRUE;
									ELSE bDoorClosingInitFlag		:= FALSE;
									END_IF
									
								ELSE
									
									bCloseDoor						:= FALSE;
									bOpenDoor						:= TRUE;
									
								END_IF
								
								IF bDoorOpened AND stProcessCylinder.Status.bReady AND stVacuumCylinder.Status.bReady THEN
									
									stProcessDoor.State				:= E_ProcessDoor_State.READY;									
									bOpenDoor						:= FALSE;
																	
								END_IF
	
	
	E_ProcessDoor_State.READY:
								
								bCloseDoor							:= FALSE;
								bOpenDoor							:= FALSE;
	
								IF stProcessDoor.CMD.bExecute AND 	stProcessDoor.CMD.ProcessDoorCMD.OpenDoor	THEN

									stProcessDoor.State				:= E_ProcessDoor_State.OPEN;
									
								ELSIF stProcessDoor.CMD.bExecute AND 	stProcessDoor.CMD.ProcessDoorCMD.CloseDoor	THEN
									
									stProcessDoor.State				:= E_ProcessDoor_State.CLOSE;									
																		
								END_IF
	

	E_ProcessDoor_State.OPEN:
	
								bOpenDoor							:= TRUE;
								
								IF bDoorOpened	THEN
									
									stProcessDoor.State				:= E_ProcessDoor_State.DONE;
								
								END_IF
								
	E_ProcessDoor_State.CLOSE:
	
								bCloseDoor							:= TRUE;
								
								IF bDoorClosed THEN
									
									stProcessDoor.State				:= E_ProcessDoor_State.DONE;
								
								END_IF
								
	E_ProcessDoor_State.DONE:
	
	
								IF stProcessDoor.CMD.bAcknowledge THEN
									
									stProcessDoor.CMD.bAcknowledge	:= FALSE;
									stProcessDoor.State				:= E_ProcessDoor_State.RESET;
								
								END_IF
	
	
	E_ProcessDoor_State.RESET:	
	
								bOpenDoor							:= FALSE;
								bCloseDoor							:= FALSE;
								
								IF NOT stProcessDoor.CMD.bAbort AND NOT stProcessDoor.CMD.bEndCycle THEN
									
									stProcessDoor.State				:= E_ProcessDoor_State.READY;
									
								ELSE stProcessDoor.State			:= E_ProcessDoor_State.ABORTED;
								END_IF
	
					
	E_ProcessDoor_State.STOPPING:					
									
								bOpenDoor							:= TRUE;
									
								IF bDoorOpened THEN
									
									bOpenDoor						:= FALSE;
									stProcessDoor.State				:= E_ProcessDoor_State.RESET;
								
								END_IF
								
							
														
									

ELSE stProcessDoor.State		:= E_ProcessDoor_State.ABORTED;
	
END_CASE
/////////////////////////////////////////////////////////////////////////////////////STATUS/////////////////////////////////////////////////////////////////////////////////////

stProcessDoor.Status.bBusy			:= 	stProcessDoor.State	= E_ProcessDoor_State.CLOSE OR
										stProcessDoor.State	= E_ProcessDoor_State.OPEN OR 
										stProcessDoor.State	= E_ProcessDoor_State.STOPPING;
								
stProcessDoor.Status.bDone			:=	stProcessDoor.State	= E_ProcessDoor_State.DONE;

stProcessDoor.Status.bReady			:= 	stProcessDoor.State	= E_ProcessDoor_State.READY;

stProcessDoor.Status.bStopped		:= 	NOT stProcessDoor.Status.bBusy;

stProcessDoor.Status.bHomed			:= 	bDoorOpened;
END_ACTION

ACTION b_ACT_IO_B:
tonDoorOpened( IN := NOT bDoorClosed, PT := stTimers.tDoorOpenedSignal);


bDoorClosed								:= dw_T05_EL1918.iProcessDoorClosed1 AND dw_T05_EL1918.iProcessDoorClosed2 AND dw_T05_EL1918.iProcessDoorFB;
bDoorOpened								:= tonDoorOpened.Q; 
bProcessDoorClosed						:= bDoorClosed;

bDoorOpenedFlag							:= bDoorOpened;

dw_T09_EL2809.qOpenProcessDoor			:= bOpenDoor OR bOpenDoorHMI OR stStationEvents[4].aEvents[0].bEventTimer.Q;//OR bOpenDoorCycleFault;	
dw_T09_EL2809.qCloseProcessDoor			:= bCloseDoor OR bCloseDoorHMI;
END_ACTION

ACTION c_Manual:


IF bProcessDoor_Down AND stTwinSAFE.qTwoHandsSafe THEN
	
	bCloseDoorHMI					:= TRUE;
	bProcessDoor_Down				:= FALSE;
	
ELSIF bDoorClosed  OR NOT stMachineStatus.bManualMode THEN

	 bCloseDoorHMI					:= FALSE;
	 bProcessDoor_Down				:= FALSE;

END_IF

IF bProcessDoor_UP THEN
	
	bOpenDoorHMI					:= TRUE;
	
	
ELSIF bDoorOpened OR  NOT stMachineStatus.bManualMode THEN

	bOpenDoorHMI					:= FALSE;	 
	
END_IF
END_ACTION

ACTION d_ACT_Set_Events_Station_4B:
//IMMEDIATE FAULTS 20..29

stStationEvents[4].aEvents[20].bEventTimer( IN :=  (bCloseDoor OR bCloseDoorHMI) AND NOT bDoorClosed, PT := T#2S);
stStationEvents[4].aEvents[20].bFault						:= TRUE;
stStationEvents[4].aEvents[20].bEventFlag					:= stStationEvents[4].aEvents[0].bEventTimer.Q;
stStationEvents[4].aEvents[20].bEventText					:= 'Process Door extend timeout';
stStationEvents[4].aEvents[20].sSolution					:= 'Check cylinder, neumatic connections and sensors';

stStationEvents[4].aEvents[21].bEventTimer( IN :=  (bOpenDoor OR bOpenDoorHMI) AND NOT bDoorOpened, PT := T#2S);
stStationEvents[4].aEvents[21].bFault						:= TRUE;
stStationEvents[4].aEvents[21].bEventFlag					:= stStationEvents[4].aEvents[1].bEventTimer.Q;
stStationEvents[4].aEvents[21].bEventText					:= 'Process Door Retract timeout';
stStationEvents[4].aEvents[21].sSolution					:= 'Check cylinder, neumatic connections and sensors';





//CYCLE STOP REQUEST 50..59

(*stStationEvents[4].aEvents[2].bCycleStopRequest			:= TRUE;
stStationEvents[4].aEvents[2].bEventFlag					:= bEventsFlag[2];
stStationEvents[4].aEvents[2].bEventText					:= 'ST1 EVENT 7';*)
END_ACTION

END_PROGRAM

// ---- POUs/B_STATIONS/B_4_PROCESS_CYLINDER__SLIDE_DOOR_VACUUM_CYLINDER/B_4_1_PRG_Master_VacuumCylinder.TcPOU
PROGRAM B_4_1_PRG_Master_VacuumCylinder

VAR

	
	
/////////////////////////////////////////////////////////////////////////////////////I O/////////////////////////////////////////////////////////////////////////////////////	
	bExtended							: ARRAY[1..2] OF BOOL;
	bRetracted							: ARRAY[1..2] OF BOOL;
	bExtend								: ARRAY[1..2] OF BOOL;
	bRetract							: ARRAY[1..2] OF BOOL;
	
	bProcessDoorClosed					: BOOL;
	
END_VAR

d_ACT_Set_Events_Station_4A();
a_ACT_Ctrl_Station_4A();
b_ACT_IO_A();

ACTION a_ACT_Ctrl_Station_4A:
/////////////////////////////////////////////////////////////////////////////////////UTILITIES/////////////////////////////////////////////////////////////////////////////////////

/////////////////////////////////////////////////////////////////////////////////////CONDITIONS/////////////////////////////////////////////////////////////////////////////////////


IF stVacuumCylinder.CMD.bAbort THEN
	
	stVacuumCylinder.State				:= E_VacuumCylinder_State.RESET;

END_IF

CASE stVacuumCylinder.State OF
	
	E_VacuumCylinder_State.ABORTED:
	
								IF stVacuumCylinder.CMD.bEnable THEN
									
									stVacuumCylinder.State				:= E_VacuumCylinder_State.HOMING;
								
								END_IF
								
	E_VacuumCylinder_State.HOMING:
	
	
								IF NOT bRetracted[1]  THEN
									
									bRetract[1]							:= TRUE;
									
								END_IF
								
								IF NOT bRetracted[2] THEN
									
									bRetract[2]							:= TRUE;
									
								END_IF
								
								
								IF bRetracted[1] AND bRetracted[2] THEN
									
									bRetract[1]							:= FALSE;
									bRetract[2]							:= FALSE;
									stVacuumCylinder.State				:= E_VacuumCylinder_State.READY;
									
								
								END_IF
	
	E_VacuumCylinder_State.READY:
	
								IF stVacuumCylinder.CMD.bExecute AND (stVacuumCylinder.CMD.VacuumCylinderCMD.Extend1 OR stVacuumCylinder.CMD.VacuumCylinderCMD.Extend2)  THEN

									stVacuumCylinder.State				:= E_VacuumCylinder_State.EXTEND;
									
								ELSIF stVacuumCylinder.CMD.bExecute AND (stVacuumCylinder.CMD.VacuumCylinderCMD.Retract1 OR stVacuumCylinder.CMD.VacuumCylinderCMD.Retract2) THEN
									
									stVacuumCylinder.State				:= E_VacuumCylinder_State.RETRACT;		
																		
								END_IF
	
	E_VacuumCylinder_State.EXTEND:
	
								bExtend[1]									:= stVacuumCylinder.CMD.VacuumCylinderCMD.Extend1;
								bExtend[2]									:= stVacuumCylinder.CMD.VacuumCylinderCMD.Extend2;
								
								IF (bExtended[1] OR NOT stVacuumCylinder.CMD.VacuumCylinderCMD.Extend1) AND (bExtended[2] OR NOT stVacuumCylinder.CMD.VacuumCylinderCMD.Extend2) THEN
									
									stVacuumCylinder.State			:= E_VacuumCylinder_State.DONE;

								END_IF
								
	E_VacuumCylinder_State.RETRACT:
	
								bRetract[1]									:= stVacuumCylinder.CMD.VacuumCylinderCMD.Retract1;
								bRetract[2]									:= stVacuumCylinder.CMD.VacuumCylinderCMD.Retract2;
								
								
								IF (bRetracted[1] OR NOT stVacuumCylinder.CMD.VacuumCylinderCMD.Retract1) AND (bRetracted[2] OR NOT stVacuumCylinder.CMD.VacuumCylinderCMD.Retract2) THEN
									
									stVacuumCylinder.State			:= E_VacuumCylinder_State.DONE;

								END_IF
								
								
	E_VacuumCylinder_State.DONE:
	
								IF stVacuumCylinder.CMD.bAcknowledge THEN
									
									stVacuumCylinder.CMD.bAcknowledge		:= FALSE;
									stVacuumCylinder.State					:= E_VacuumCylinder_State.RESET;
								
								END_IF
	
	
	E_VacuumCylinder_State.RESET:	
	
								bExtend[1]									:= FALSE;								
								bRetract[1]									:= FALSE;
								bExtend[2]									:= FALSE;								
								bRetract[2]									:= FALSE;
								
								IF NOT stVacuumCylinder.CMD.bAbort AND NOT stVacuumCylinder.CMD.bEndCycle THEN
									
									stVacuumCylinder.State					:= E_VacuumCylinder_State.READY;
									
								ELSE stVacuumCylinder.State					:= E_VacuumCylinder_State.ABORTED;
								END_IF
									

ELSE stVacuumCylinder.State	:= E_VacuumCylinder_State.ABORTED;
	
END_CASE
/////////////////////////////////////////////////////////////////////////////////////STATUS/////////////////////////////////////////////////////////////////////////////////////

stVacuumCylinder.Status.bBusy		:= 	stVacuumCylinder.State	= E_VacuumCylinder_State.EXTEND OR
										stVacuumCylinder.State	= E_VacuumCylinder_State.RETRACT OR 
										stVacuumCylinder.State	= E_VacuumCylinder_State.STOPPING;
								
stVacuumCylinder.Status.bDone		:=	stVacuumCylinder.State	= E_VacuumCylinder_State.DONE;

stVacuumCylinder.Status.bReady		:= 	stVacuumCylinder.State	= E_VacuumCylinder_State.READY;

stVacuumCylinder.Status.bStopped	:= 	NOT stVacuumCylinder.Status.bBusy;

stVacuumCylinder.Status.bHomed		:= 	bRetracted[1] AND bRetracted[2];
END_ACTION

ACTION b_ACT_IO_A:

bExtended[1]								:= dw_T08_EL1809.iVacuumCylinderExtended1;
bRetracted[1]								:= dw_T08_EL1809.iVacuumCylinderRetracted1;
bExtended[2]								:= dw_T08_EL1809.iVacuumCylinderExtended2;
bRetracted[2]								:= dw_T08_EL1809.iVacuumCylinderRetracted2;




IF (bExtend[1] OR bVacuumCylinderExtend1) AND bProcessDoorClosed  THEN
	
	dw_T09_EL2809.qExtendVacuumCylinder1	:= TRUE ;
	dw_T09_EL2809.qRetractVacuumCylinder1	:= FALSE;

ELSIF (bRetract[1] OR bVacuumCylinderRetract1)  THEN
	
	dw_T09_EL2809.qExtendVacuumCylinder1	:= FALSE;
	dw_T09_EL2809.qRetractVacuumCylinder1	:= TRUE;
	
ELSIF stMachineStatus.bFault THEN
	
	dw_T09_EL2809.qExtendVacuumCylinder1	:= FALSE;
	dw_T09_EL2809.qRetractVacuumCylinder1	:= FALSE;

END_IF

IF (bExtend[2] OR bVacuumCylinderExtend2)  AND bProcessDoorClosed  THEN
	
	dw_T10_EL2809.qExtendVacuumCylinder2	:= TRUE ;
	dw_T10_EL2809.qRetractVacuumCylinder2	:= FALSE;

ELSIF (bRetract[2] OR bVacuumCylinderRetract2)  THEN
	
	dw_T10_EL2809.qExtendVacuumCylinder2	:= FALSE;
	dw_T10_EL2809.qRetractVacuumCylinder2	:= TRUE;
	
ELSIF stMachineStatus.bFault THEN
	
	dw_T10_EL2809.qExtendVacuumCylinder2	:= FALSE;
	dw_T10_EL2809.qRetractVacuumCylinder2	:= FALSE;

END_IF


bProcessDoorClosed := dw_T05_EL1918.iProcessDoorClosed1 AND dw_T05_EL1918.iProcessDoorClosed2 AND dw_T05_EL1918.iProcessDoorFB;

bEnable_VacuumCylinder[1]					:= bPartHeld[1];
bEnable_VacuumCylinder[2]					:= bPartHeld[2];
END_ACTION

ACTION d_ACT_Set_Events_Station_4A:
//FAULTS 10..19

stStationEvents[4].aEvents[10].bEventTimer( IN := (bExtend[1] AND NOT bExtended[1]), PT := T#3S);
stStationEvents[4].aEvents[10].bFault						:= TRUE;
stStationEvents[4].aEvents[10].bEventFlag					:= stStationEvents[3].aEvents[0].bEventTimer.Q;
stStationEvents[4].aEvents[10].bEventText					:= 'Vacuum Cylinder 1 extend timeout';
stStationEvents[4].aEvents[10].sSolution						:= 'Check cylinder, neumatic connections and sensors';

stStationEvents[4].aEvents[11].bEventTimer( IN := (bRetract[1] AND NOT bRetracted[1]), PT := T#3S);
stStationEvents[4].aEvents[11].bFault						:= TRUE;
stStationEvents[4].aEvents[11].bEventFlag					:= stStationEvents[3].aEvents[1].bEventTimer.Q;
stStationEvents[4].aEvents[11].bEventText					:= 'Vacuum Cylinder retract timeout';
stStationEvents[4].aEvents[11].sSolution						:= 'Check cylinder, neumatic connections and sensors';

stStationEvents[4].aEvents[12].bEventTimer( IN := (bExtend[2] AND NOT bExtended[2]), PT := T#3S);
stStationEvents[4].aEvents[12].bFault						:= TRUE;
stStationEvents[4].aEvents[12].bEventFlag					:= stStationEvents[3].aEvents[2].bEventTimer.Q;
stStationEvents[4].aEvents[12].bEventText					:= 'Vacuum Cylinder 2 extend timeout';
stStationEvents[4].aEvents[12].sSolution						:= 'Check cylinder, neumatic connections and sensors';

stStationEvents[4].aEvents[13].bEventTimer( IN := (bRetract[2] AND NOT bRetracted[2]), PT := T#3S);
stStationEvents[4].aEvents[13].bFault						:= TRUE;
stStationEvents[4].aEvents[13].bEventFlag					:= stStationEvents[3].aEvents[3].bEventTimer.Q;
stStationEvents[4].aEvents[13].bEventText					:= 'Vacuum Cylinder retract timeout';
stStationEvents[4].aEvents[13].sSolution						:= 'Check cylinder, neumatic connections and sensors';


//CYCLE STOP REQUEST 40..49

(*stStationEvents[3].aEvents[2].bCycleStopRequest			:= TRUE;
stStationEvents[3].aEvents[2].bEventFlag					:= ;
stStationEvents[3].aEvents[2].bEventText					:= 'ST1 EVENT 7';*)
END_ACTION

END_PROGRAM

// ---- POUs/A_MASTER/A_2_PRG_MachineCtrl.TcPOU
PROGRAM A_2_PRG_MachineCtrl
VAR
/////////////////////////////////////////////////////////////////////////////////////TIMERS & TRIGGERS/////////////////////////////////////////////////////////////////////////////////////

	tonSys_Init					: Tc2_Standard.TON:=(PT:=T#1S);
	tonSys_InitTimeout			: Tc2_Standard.TON:=(PT:=T#15S);					
	tonFirstAutoCycle			: Tc2_Standard.TON:=(PT:=T#500MS);
	tonStopped					: TON := (PT := T#500MS);
	rStartConditionTrigger		: R_TRIG;
	tonNoPartPresent			: TON;
	
/////////////////////////////////////////////////////////////////////////////////////PROCESS CYCLE/////////////////////////////////////////////////////////////////////////////////////	
	
	eCycleState					: E_General_ProcessCycle;
	tonCMD_Done					: TON;
	tonResetAllCMD				: TON;
	tonExecute					: TON;
	tonSave_Data				: TON;
	tonWriteToCsv				: TON;
	rFirstAutoCycle				: R_TRIG;
	
	bStartProcessCondition		: BOOL;
	bLeakTestDoneFlag			: BOOL;
	bHeightTestDoneFlag			: BOOL;
	i							: INT;

	tonGettingResults			: TON;
	ctuRejectPart				: CTU;
	
/////////////////////////////////////////////////////////////////////////////////////I/O/////////////////////////////////////////////////////////////////////////////////////	

	rRejectSensor				: R_TRIG;
	bTwoHandsSignal				: BOOL;
	tonTwoHandsSignal			: TON;
	
	bProcessedPart				: ARRAY[0..1] OF BOOL;
	
		(* Renan Added - Buglist n6 - 08Jul26 *)
	bNest1StartOK				: BOOL;
	bNest2StartOK				: BOOL;
	bCycleHasFailure 			: BOOL;
	bCycleAllProcessedPass		: BOOL;
	(*\Renan Added - Buglist n6 - 08Jul26 *)
	
	bPuckLockerReadyToStart		: BOOL; (* Renan Added - Puck Locker Bug - 08Jul26 *)
	nPucksToRelease 			: USINT;(* Renan Added - Puck Locker Bug - 08Jul26 *)
	bPuckLockerEnable       	: BOOL; (* Renan added - Puck Locker Bug - 10Jul26*)
	
	//General Dtation CMD
	
	bGeneralEnable				: BOOL;
	bGeneralRST					: BOOL;
	bGeneralAbort				: BOOL;
	bGeneralManualMode			: BOOL;
	
	
END_VAR

/////////////////////////////////////////////////////////////////////////////////////GENERAL/////////////////////////////////////////////////////////////////////////////////////
a_ACT_MachineStatus();
b_ACT_ProcessCycle();
d_ACT_IO();

ACTION a_ACT_MachineStatus:
/////////////////////////////////////////////////////////////////////////////////////Utilities/////////////////////////////////////////////////////////////////////////////////////
tonSys_Init(IN:=stMachineStatus.bInitialising);
tonSys_InitTimeout(IN:=stMachineStatus.bInitialising);
tonSafety( IN := stMachineStatus.eMachineState = E_MachineState.SAFETY, PT := T#10S);
tonStopped(IN := stMachineStatus.eMachineState = E_MachineState.STOPPED);
	
	IF stMachineStatus.eMachineState <> E_MachineState.SYSTEM_AUTO_CYCLE AND 
		stMachineStatus.eMachineState <> E_MachineState.SYSTEM_INITIALISING THEN
		
		sMachineMessage									:= '';			
		
	END_IF
	
	IF (stMachineStatus.eMachineState = E_MachineState.STOPPED)  OR 
		(stMachineStatus.eMachineState = E_MachineState.STOPPING) THEN
		
		stTwinSAFE.iMachineStopped						:= TRUE;
		stTwinSAFE.iRunSafety							:= FALSE;
	
	ELSIF (stMachineStatus.eMachineState = E_MachineState.SAFETY) OR (stMachineStatus.eMachineState = E_MachineState.SYSTEM_INITIALISING) OR 
		(stMachineStatus.eMachineState = E_MachineState.SYSTEM_READY_TO_START) OR (stMachineStatus.eMachineState = E_MachineState.SYSTEM_AUTO_CYCLE) 
		OR (stMachineStatus.eMachineState = E_MachineState.MANUAL_MODE)THEN

		stTwinSAFE.iRunSafety							:= TRUE;
		stTwinSAFE.iMachineStopped						:= FALSE;
	
	ELSE stTwinSAFE.iMachineStopped						:= FALSE;
		stTwinSAFE.iRunSafety							:= FALSE;
		
	END_IF
	
	IF stMachineStatus.eMachineState = E_MachineState.SAFETY THEN
		
		stTwinSAFE.iInitSafety							:= TRUE;
		
	ELSE stTwinSAFE.iInitSafety							:= FALSE;
		
	END_IF

/////////////////////////////////////////////////////////////////////////////////////CONDITIONS/////////////////////////////////////////////////////////////////////////////////////
				IF NOT stMasterCtrl.bNoFault THEN
					stMachineStatus.eMachineState 		:= E_MachineState.FAULT;
				END_IF
				
				IF stMachineStatus.eMachineState		= E_MachineState.STOPPING OR
				stMachineStatus.eMachineState			= E_MachineState.FAULT THEN
					
					bGeneralAbort						:= TRUE;
					
					bGeneralEnable						:= FALSE;
					
				END_IF
				
				IF 	stButtonsLamps.bResetButtonFallingEdge THEN
					
					bGeneralRST							:= TRUE;
					
				ELSE 
					
					bGeneralRST							:= FALSE;
					
				END_IF	

				IF 	NOT (stMachineStatus.eMachineState = E_MachineState.MANUAL_MODE) THEN
					
					bGeneralManualMode					:= FALSE;
					
				END_IF
				
				IF stMachineStatus.eMachineState = E_MachineState.SYSTEM_POWER_UP THEN
					
					bReadAMSNetID						:= TRUE;
				
				ELSE 
					
					bReadAMSNetID						:= FALSE;
					
				END_IF
				
				IF stMachineStatus.eMachineState		= E_MachineState.FAULT THEN
					
					bOpenDoorCycleFault					:= TRUE;
					
				ELSE bOpenDoorCycleFault				:= FALSE;
					
				END_IF
				
/////////////////////////////////////////////////////////////////////////////////////MACHINE CONTROL/////////////////////////////////////////////////////////////////////////////////////

CASE stMachineStatus.eMachineState OF

E_MachineState.SYSTEM_POWER_UP: 		

				fbGetLocalAMSNetID.bExecute				:= TRUE;
				bLightsOnOff							:= TRUE;
				IF tonSystemPowerUP.Q THEN
						stMachineStatus.eMachineState 	:= E_MachineState.STOPPED;//
				END_IF
	
E_MachineState.STOPPED:		

				stTwinSAFE.iRunSafety					:= FALSE;				

				IF stMasterCtrl.bNoFault   AND NOT stMasterCtrl.bCycleStopRequest AND ftrigButton[3].Q AND tonStopped.Q THEN
						stMachineStatus.eMachineState 	:= E_MachineState.SAFETY;//
				ELSIF NOT stMasterCtrl.bNoFault    THEN	
					stMachineStatus.eMachineState 		:= E_MachineState.FAULT;		
				END_IF	

E_MachineState.SAFETY:

				GVL_IO.dw_T09_EL2809.qOpenProcessDoor   := TRUE; 
				stTwinSAFE.iRunSafety					:= TRUE;
				
				IF stTwinSAFE.qSafetyOk THEN
					
					stMachineStatus.eMachineState		:= E_MachineState.SYSTEM_INITIALISING;
					
				ELSIF stButtonsLamps.bStopButtonFallingEdge OR  
				stMasterCtrl.bCycleStopRequest OR tonSys_InitTimeout.Q  THEN
				
					stMachineStatus.eMachineState 		:= E_MachineState.STOPPING;	
					
				ELSIF NOT stMasterCtrl.bNoFault THEN		
					
					stMachineStatus.eMachineState 		:= E_MachineState.FAULT;
	
				END_IF
								

E_MachineState.SYSTEM_INITIALISING:		
					
				bGeneralAbort							:= FALSE;		

				IF NOT stProcessCylinder.Status.bHomed OR NOT stVacuumCylinder.Status.bHomed THEN
						
						sMachineMessage					:= 'trigger both safety buttons to reset machine';
						
						IF bTwoHandsSignal THEN
							
							tonSys_InitTimeout.IN		:= TRUE;
							
							bGeneralEnable				:= TRUE;
							sMachineMessage				:= '';
							
						END_IF
				ELSIF stProcessCylinder.Status.bHomed AND stVacuumCylinder.Status.bHomed  THEN
					
							bGeneralEnable				:= TRUE;				
				
				END_IF
				
				IF stMasterCtrl.bAllStationsReady  THEN 
					stMachineStatus.eMachineState		:= E_MachineState.SYSTEM_READY_TO_START;
				ELSIF stButtonsLamps.bStopButtonFallingEdge OR  
				stMasterCtrl.bCycleStopRequest OR tonSys_InitTimeout.Q  THEN
					stMachineStatus.eMachineState 		:= E_MachineState.STOPPING;	
				ELSIF NOT stMasterCtrl.bNoFault THEN		
					stMachineStatus.eMachineState 		:= E_MachineState.FAULT;
				END_IF
			
					
E_MachineState.SYSTEM_READY_TO_START:	

				IF 	 stButtonsLamps.bStartButtonFallingEdge AND stMasterCtrl.bAllStationsReady  THEN
					stMachineStatus.eMachineState 		:= E_MachineState.SYSTEM_AUTO_CYCLE;
				ELSIF NOT stMasterCtrl.bAllStationsReady OR stMasterCtrl.bCycleStopRequest THEN
					stMachineStatus.eMachineState 		:= E_MachineState.STOPPING;		
				ELSIF NOT stMasterCtrl.bNoFault THEN	
					stMachineStatus.eMachineState 		:= E_MachineState.FAULT;
				ELSIF GVL_Master.stMasterCTRL.bManualModeRequest AND stMasterCtrl.bNoFault THEN
					stMachineStatus.eMachineState 		:= E_MachineState.MANUAL_MODE;
				END_IF

				

E_MachineState.SYSTEM_AUTO_CYCLE:		

				
				IF  stMasterCtrl.bCycleStopRequest AND (eCycleState = E_General_ProcessCycle.IDLE) THEN
	
					stMachineStatus.eMachineState 		:= E_MachineState.STOPPING;
				
				ELSIF stMasterCtrl.bCycleStopRequest AND NOT (eCycleState = E_General_ProcessCycle.IDLE) THEN					
				
					sMachineMessage						:= 'Ending  Cycle';
				
				ELSIF NOT stMasterCtrl.bNoFault THEN	
					stMachineStatus.eMachineState 		:= E_MachineState.FAULT;
				END_IF
				

E_MachineState.STOPPING:	

				
				IF stMasterCtrl.bAllStationsStopped THEN
					stMachineStatus.eMachineState 		:= E_MachineState.STOPPED;
				ELSIF NOT stMasterCtrl.bNoFault THEN	
					stMachineStatus.eMachineState 		:= E_MachineState.FAULT;					
				END_IF
				
				stTwinSAFE.iRunSafety					:= FALSE;	

E_MachineState.FAULT:	
				
				GVL_IO.dw_T09_EL2809.qOpenProcessDoor   :=TRUE; // Thays added - Buglist n1 - 08Jul26

				IF stMasterCtrl.bNoFault	THEN
					stMachineStatus.eMachineState		:= E_MachineState.STOPPED;		
				END_IF
				
				stTwinSAFE.iRunSafety					:= FALSE;	

E_MachineState.MANUAL_MODE:

				IF stButtonsLamps.bStopButtonFallingEdge OR NOT GVL_Master.stMasterCTRL.bManualModeRequest THEN
					stMachineStatus.eMachineState 		:= E_MachineState.STOPPING;
				ELSIF  NOT stMasterCtrl.bNoFault THEN	
					stMachineStatus.eMachineState 		:= E_MachineState.FAULT;								
				ELSE 
					
					bGeneralManualMode					:=TRUE;

				END_IF
				
					
ELSE
stMachineStatus.eMachineState:=E_MachineState.SYSTEM_POWER_UP;		
END_CASE									


/////////////////////////////////////////////////////////////////////////////////////MACHINE STATUS/////////////////////////////////////////////////////////////////////////////////////
stMachineStatus.bSystemPowerUp 			:= (stMachineStatus.eMachineState = E_MachineState.SYSTEM_POWER_UP);
stMachineStatus.bStopped 				:= (stMachineStatus.eMachineState = E_MachineState.STOPPED);
stMachineStatus.bInitialising 			:= (stMachineStatus.eMachineState = E_MachineState.SYSTEM_INITIALISING);
stMachineStatus.bReadyToStart 			:= (stMachineStatus.eMachineState = E_MachineState.SYSTEM_READY_TO_START);
stMachineStatus.bAutoCycle 				:= (stMachineStatus.eMachineState = E_MachineState.SYSTEM_AUTO_CYCLE);
stMachineStatus.bStopping 				:= (stMachineStatus.eMachineState = E_MachineState.STOPPING);
stMachineStatus.bFault 					:= (stMachineStatus.eMachineState = E_MachineState.FAULT);
stMachineStatus.bManualMode 			:= (stMachineStatus.eMachineState = E_MachineState.MANUAL_MODE);
stMachineStatus.bSafety 				:= (stMachineStatus.eMachineState = E_MachineState.SAFETY);

/////////////////////////////////////////////////////////////////////////////////////FLAGS/////////////////////////////////////////////////////////////////////////////////////
stMasterCtrl.bAllStationsStopped		:= (*stLSS.Status.bStopped AND*) stLeakTesters.Status.bStopped AND stProcessCylinder.Status.bStopped AND stProcessDoor.Status.bStopped AND stVacuumCylinder.Status.bStopped AND
										   NOT stLSS.Status.bBusy AND NOT stLeakTesters.Status.bBusy  AND NOT stProcessCylinder.Status.bBusy AND NOT stProcessDoor.Status.bBusy AND NOT stVacuumCylinder.Status.bBusy;
										   
stMasterCtrl.bAllStationsReady			:= (*stLSS.Status.bReady  AND*) stLeakTesters.Status.bReady AND stCamera.Status.bReady AND stProcessCylinder.Status.bReady AND stProcessDoor.Status.bReady AND stVacuumCylinder.StatuS.bReady;
END_ACTION

ACTION b_ACT_ProcessCycle:
/////////////////////////////////////////////////////////////////////////////////////UTILITIES & TRIGGERS/////////////////////////////////////////////////////////////////////////////////////
//ADD REJECT SENSOR FUNCTION. IF PART FAIL WE SHOULD WAIT UNTIL THE OPERATOR LEAVE THE FAIL PART IN THE CONTAINER

tonNoPartPresent(PT := T#2S);

ctuRejectPart();
IF eCycleState = E_General_ProcessCycle.RESET_ALL_CMD THEN
	
	ctuRejectPart.RESET															:= TRUE;

ELSE ctuRejectPart.RESET														:= FALSE;	
	
END_IF
IF eCycleState = E_General_ProcessCycle.IDLE THEN
	
	bAutocycleIDLE																:= TRUE;
	
ELSE bAutocycleIDLE																:= FALSE;

END_IF

tonGettingResults( IN := eCycleState = E_General_ProcessCycle.WAIT_RESULTS, PT := T#100MS);

tonCMD_Done( IN := , PT := T#500MS);
tonSave_Data( IN :=  eCycleState = E_General_ProcessCycle.SAVE_DATA2, PT := T#500MS);
tonResetAllCMD( IN := eCycleState = E_General_ProcessCycle.RESET_ALL_CMD, PT := T#500MS);


tonExecute( IN := 	eCycleState = E_General_ProcessCycle.CLOSE_PROCESS_DOOR OR
					eCycleState = E_General_ProcessCycle.OPEN_PROCESS_DOOR OR
					eCycleState = E_General_ProcessCycle.EXTEND_PROCESS_CYLINDER OR
					eCycleState = E_General_ProcessCycle.RETRACT_PROCESS_CYLINDER OR
					eCycleState = E_General_ProcessCycle.HOLD_PART OR
					eCycleState = E_General_ProcessCycle.RELEASE_PART OR
					eCycleState = E_General_ProcessCycle.LEAK_TEST_HEIGHT_CHECK OR
					eCycleState = E_General_ProcessCycle.CAMERA_CHECK_PART_PRESENT OR
					eCycleState = E_General_ProcessCycle.VACUUM_CYLINDER_EXTENSION OR
					eCycleState = E_General_ProcessCycle.VACUUM_CYLINDER_RETRACTION OR
					eCycleState = E_General_ProcessCycle.WAIT_TO_SAVE_DATA,
					PT := T#500MS);
					
IF (stMachineStatus.eMachineState <> E_MachineState.SYSTEM_AUTO_CYCLE) THEN
	
	eCycleState																	:= E_General_ProcessCycle.RESET_ALL_CMD;

END_IF

rFirstAutoCycle( CLK := stMachineStatus.bAutoCycle);

IF (eCycleState = E_General_ProcessCycle.LEAK_TEST_HEIGHT_CHECK) OR (eCycleState = E_General_ProcessCycle.WAIT_LEAK_TEST_HEIGHT_CHECK) THEN
	
			sMachineMessage														:= 'Inspection in process ';

END_IF

IF stMachineStatus.eMachineState <> E_MachineState.SYSTEM_AUTO_CYCLE THEN
	
	MEMSET( destAddr := ADR(stCycleDataNest1), fillByte := 0, n := SIZEOF(stCycleDataNest1));
	MEMSET( destAddr := ADR(stCycleDataNest2), fillByte := 0, n := SIZEOF(stCycleDataNest2));

END_IF

(* Renan Added 10Jul26*)
bPuckLockerEnable := GVL_HMI.bPuckLockerGateEnable;
(*\Renan Added 10Jul26*)

(*Renan added - Puck Locker Bug - 08Jul26*)
bPuckLockerReadyToStart := (NOT bPuckLockerEnable) OR (GVL_Stations.stPuckLocker.bPuckDetected AND
							GVL_Stations.stPuckLocker.bPuckLocked AND GVL_Stations.stPuckLocker.eState = E_PuckLockerState.Locked);
(*\Renan added - Puck Locker Bug - 08Jul26*)

(*Renan Added 06Jul26*)
IF bPuckLockerEnable THEN
	GVL_Stations.stPuckLocker.bNestsEmpty := ((NOT bProcessedPart[0]) OR (NOT bPartPresentNest1)) AND ((NOT bProcessedPart[1]) OR (NOT bPartPresentNest2));
ELSE
	GVL_Stations.stPuckLocker.bNestsEmpty := TRUE;
END_IF
(*\Renan Added 06Jul26*)

	
/////////////////////////////////////////////////////////////////////////////////////CONDITIONS/////////////////////////////////////////////////////////////////////////////////////

(* Renan Added - Buglist n6 - 08Jul26 *)
bNest1StartOK := (NOT bNest1Flag) OR bPartPresentNest1;
bNest2StartOK := (NOT bNest2Flag) OR bPartPresentNest2;
(*\Renan Added - Buglist n6 - 08Jul26 *)

bStartProcessCondition := (bTwoHandsSignal AND (bNest1Flag OR bNest2Flag));
rStartConditionTrigger( CLK := bStartProcessCondition);


IF rFirstAutoCycle.Q THEN
	eCycleState																	:= E_General_ProcessCycle.RESET_ALL_CMD;
END_IF


CASE eCycleState OF
	
E_General_ProcessCycle.RESET_ALL_CMD:

				stProcessDoor.CMD.ProcessDoorCMD.OpenDoor						:= FALSE;
				stProcessDoor.CMD.ProcessDoorCMD.CloseDoor						:= FALSE;
				stProcessDoor.CMD.bExecute										:= FALSE;
				stProcessDoor.CMD.bAcknowledge									:= FALSE;
				
				stProcessCylinder.CMD.ProcessCylinderCMD.ExtendCylinder1		:= FALSE;
				stProcessCylinder.CMD.ProcessCylinderCMD.RetractCylinder1		:= FALSE;
				stProcessCylinder.CMD.ProcessCylinderCMD.ExtendPartHolder1		:= FALSE;
				stProcessCylinder.CMD.ProcessCylinderCMD.RetractPartHolder1		:= FALSE;
				stProcessCylinder.CMD.bAcknowledge								:= FALSE;
				
				stProcessCylinder.CMD.ProcessCylinderCMD.ExtendCylinder2		:= FALSE;
				stProcessCylinder.CMD.ProcessCylinderCMD.RetractCylinder2		:= FALSE;
				stProcessCylinder.CMD.ProcessCylinderCMD.ExtendPartHolder2		:= FALSE;
				stProcessCylinder.CMD.ProcessCylinderCMD.RetractPartHolder2		:= FALSE;
				
				stProcessCylinder.CMD.bExecute									:= FALSE;
				
				stVacuumCylinder.CMD.VacuumCylinderCMD.Extend1					:= FALSE;
				stVacuumCylinder.CMD.VacuumCylinderCMD.Retract1					:= FALSE;
				stVacuumCylinder.CMD.VacuumCylinderCMD.Extend2					:= FALSE;
				stVacuumCylinder.CMD.VacuumCylinderCMD.Retract2					:= FALSE;
				stVacuumCylinder.CMD.bExecute									:= FALSE;
				stVacuumCylinder.CMD.bAcknowledge								:= FALSE;
				
				stLeakTesters.CMD.LeakTestersCMD.RunLeakTester1					:= FALSE;
				stLeakTesters.CMD.LeakTestersCMD.RunLeakTester2					:= FALSE;
				stLeakTesters.CMD.bExecute										:= FALSE;
				stLeakTesters.CMD.bAcknowledge									:= FALSE;
				
				stLSS.CMD.LSS_CMD.Measurement1									:= FALSE;
				stLSS.CMD.LSS_CMD.Measurement1									:= FALSE;
				stLSS.CMD.bExecute												:= FALSE;
				stLSS.CMD.bAcknowledge											:= FALSE;
				
				stCamera.CMD.bExecute											:= FALSE;
				stCamera.CMD.CameraCMD.Inspect1									:= FALSE;
				stCamera.CMD.CameraCMD.Inspect2									:= FALSE;
				stCamera.CMD.CameraCMD.PartPresent1								:= FALSE;
				stCamera.CMD.CameraCMD.PartPresent2								:= FALSE;
				stCamera.CMD.CameraCMD.ContinuousPartPresent1					:= FALSE;
				stCamera.CMD.CameraCMD.ContinuousPartPresent2					:= FALSE;
				stCamera.CMD.bAcknowledge										:= FALSE;
				
				
				bWriteNest1														:= FALSE;
				bWriteNest2														:= FALSE;
				bRejectPartDialog[0]											:= FALSE;
				bRejectPartDialog[1]											:= FALSE;
				bRejectPartFault												:= FALSE;
				
				bHeightTestDoneFlag												:= FALSE;
				bLeakTestDoneFlag												:= FALSE;
				
				bProcessedPart[0]												:= FALSE;
				bProcessedPart[1]												:= FALSE;
				
				bPartPresentNest1 												:= FALSE;
				bPartPresentNest2 												:= FALSE;
				
				tonNoPartPresent.IN												:= FALSE;
			
				//add reset command to reset all cycle data
				
				IF tonResetAllCMD.Q AND stMachineStatus.bAutoCycle THEN
					
					eCycleState													:= E_General_ProcessCycle.IDLE;		
				
				END_IF
	
E_General_ProcessCycle.IDLE:
		
				sMachineMessage := 'Place Parts in the nests';
				
				//start cycle
				IF rStartConditionTrigger.Q AND NOT bProcessedPart[0] AND NOT bProcessedPart[1] AND bPuckLockerReadyToStart THEN (*Renan added - Puck Locker Bug - 08Jul26*) //Original: IF bStartProcessCondition AND NOT bProcessedPart[0] AND NOT bProcessedPart[1] THEN
					
					MEMSET( destAddr := ADR(stCycleDataNest1), fillByte := 0, n := SIZEOF(stCycleDataNest1));
					MEMSET( destAddr := ADR(stCycleDataNest2), fillByte := 0, n := SIZEOF(stCycleDataNest2));
					
					eCycleState													:= E_General_ProcessCycle.CAMERA_CHECK_PART_PRESENT;
					
				END_IF
				
				
				IF bPuckLockerEnable AND NOT bPuckLockerReadyToStart AND NOT bProcessedPart[0] AND NOT bProcessedPart[1] THEN
				
					IF NOT GVL_Stations.stPuckLocker.bPuckDetected THEN
						
						sMachineMessage 		:= 'Insert puck into locker to continue';
						
					ELSE
						
						sMachineMessage := 'Waiting for puck locker to lock puck';
						
					END_IF					
				
				ELSIF  bPuckLockerReadyToStart THEN
					
					sMachineMessage := 'trigger both safety buttons to start cycle';
						
				END_IF
			
				
E_General_ProcessCycle.CAMERA_CHECK_PART_PRESENT: 

				
				stCamera.CMD.CameraCMD.PartPresent1								:= bNest1Flag;
				stCamera.CMD.CameraCMD.PartPresent2								:= bNest2Flag;
				stCamera.CMD.bExecute											:= TRUE;
				
				IF tonExecute.Q THEN
					eCycleState													:= E_General_ProcessCycle.WAIT_CAMERA_CHECK_PART_PRESENT;	
				END_IF
				
E_General_ProcessCycle.WAIT_CAMERA_CHECK_PART_PRESENT: 
	
						
				IF stCamera.Status.bDone THEN
					
				stCamera.CMD.CameraCMD.PartPresent1								:= FALSE;
				stCamera.CMD.CameraCMD.PartPresent2								:= FALSE;
				stCamera.CMD.bExecute											:= FALSE;
				stCamera.CMD.bAcknowledge										:= TRUE;

				eCycleState														:= E_General_ProcessCycle.PART_PRESENT_CHECK;				
				
				END_IF	

E_General_ProcessCycle.PART_PRESENT_CHECK:

				IF (bPartPresentNest1 OR NOT bNest1Flag) AND (bPartPresentNest2 OR NOT bNest2Flag ) THEN
					
					IF bNest1Flag THEN
						
						bProcessedPart[0]										:= TRUE;
						
					END_IF
					
					IF bNest2Flag THEN
						
						bProcessedPart[1]										:= TRUE;
						
					END_IF
					
					eCycleState													:= E_General_ProcessCycle.CLOSE_PROCESS_DOOR;	
					
				ELSE
					
					tonNoPartPresent.IN											:= TRUE;
					
					IF (NOT bPartPresentNest1 AND bNest1Flag) AND (bPartPresentNest2 OR NOT bNest2Flag) THEN
						
						sMachineMessage 										:= 'No part Present in Nest LH';
						
					ELSIF (bPartPresentNest1 OR NOT bNest1Flag) AND ( NOT bPartPresentNest2 AND bNest2Flag) THEN
						
						sMachineMessage 										:= 'No part Present in Nest RH';
						
					ELSIF (NOT bPartPresentNest1 AND bNest1Flag) AND ( NOT bPartPresentNest2 AND bNest2Flag) THEN
						
						sMachineMessage 										:= 'No part Present in both Nests';
						
					END_IF
					
					IF tonNoPartPresent.Q THEN
						
						eCycleState												:= E_General_ProcessCycle.RESET_ALL_CMD;
						
					END_IF
					

				END_IF
			
E_General_ProcessCycle.CLOSE_PROCESS_DOOR:
				
				stProcessDoor.CMD.ProcessDoorCMD.CloseDoor						:= TRUE;
				stProcessDoor.CMD.bExecute										:= TRUE;
				
				IF tonExecute.Q THEN
					
					eCycleState													:= E_General_ProcessCycle.WAIT_CLOSE_PROCESS_DOOR;	
					
				END_IF

E_General_ProcessCycle.WAIT_CLOSE_PROCESS_DOOR:
				
				IF stProcessDoor.Status.bDone THEN
					
				stProcessDoor.CMD.ProcessDoorCMD.CloseDoor						:= FALSE;
				stProcessDoor.CMD.bExecute										:= FALSE;
				stProcessDoor.CMD.bAcknowledge									:= TRUE;
				
				eCycleState														:= E_General_ProcessCycle.EXTEND_PROCESS_CYLINDER;
				
				END_IF
					
								
E_General_ProcessCycle.EXTEND_PROCESS_CYLINDER:
				
						
				stProcessCylinder.CMD.ProcessCylinderCMD.ExtendCylinder1		:= bProcessedPart[0];
				stProcessCylinder.CMD.ProcessCylinderCMD.ExtendCylinder2		:= bProcessedPart[1];
				stProcessCylinder.CMD.bExecute									:= TRUE;
	
				IF tonExecute.Q THEN
					
					eCycleState													:= E_General_ProcessCycle.WAIT_EXTEND_PROCESS_CYLINDER;	
					
				END_IF

E_General_ProcessCycle.WAIT_EXTEND_PROCESS_CYLINDER:
			
				IF stProcessCylinder.Status.bDone THEN
					
					stProcessCylinder.CMD.ProcessCylinderCMD.ExtendCylinder1	:= FALSE;
					stProcessCylinder.CMD.ProcessCylinderCMD.ExtendCylinder2	:= FALSE;
					stProcessCylinder.CMD.bExecute								:= FALSE;
					stProcessCylinder.CMD.bAcknowledge							:= TRUE;	

					eCycleState													:= E_General_ProcessCycle.HOLD_PART;				
						
				END_IF
				
E_General_ProcessCycle.HOLD_PART:

				stProcessCylinder.CMD.ProcessCylinderCMD.ExtendPartHolder1		:= bProcessedPart[0];
				stProcessCylinder.CMD.ProcessCylinderCMD.ExtendPartHolder2		:= bProcessedPart[1];
				stProcessCylinder.CMD.bExecute									:= TRUE;
				
				IF tonExecute.Q THEN
					
					eCycleState													:= E_General_ProcessCycle.WAIT_HOLD_PART;	
					
				END_IF
				
E_General_ProcessCycle.WAIT_HOLD_PART:
			   
				IF stProcessCylinder.Status.bDone THEN
					
					stProcessCylinder.CMD.ProcessCylinderCMD.ExtendPartHolder1	:= FALSE;
					stProcessCylinder.CMD.ProcessCylinderCMD.ExtendPartHolder2	:= FALSE;
					stProcessCylinder.CMD.bExecute								:= FALSE;
					stProcessCylinder.CMD.bAcknowledge							:= TRUE;

								
					eCycleState  												:=E_General_ProcessCycle.VACUUM_CYLINDER_EXTENSION;	
						
				END_IF
				
E_General_ProcessCycle.VACUUM_CYLINDER_EXTENSION:

				stVacuumCylinder.CMD.VacuumCylinderCMD.Extend1					:= bProcessedPart[0];
				stVacuumCylinder.CMD.VacuumCylinderCMD.Extend2					:= bProcessedPart[1];
				stVacuumCylinder.CMD.bExecute									:= TRUE;
					
				IF tonExecute.Q THEN
					
					eCycleState													:= E_General_ProcessCycle.WAIT_VACUUM_CYLINDER_EXTENSION;	
					
				END_IF

E_General_ProcessCycle.WAIT_VACUUM_CYLINDER_EXTENSION:

				IF stVacuumCylinder.Status.bDone THEN
					
					stVacuumCylinder.CMD.VacuumCylinderCMD.Extend1				:= FALSE;
					stVacuumCylinder.CMD.VacuumCylinderCMD.Extend2				:= FALSE;
					stVacuumCylinder.CMD.bExecute								:= FALSE;
					stVacuumCylinder.CMD.bAcknowledge 							:= TRUE;	
					
					eCycleState													:= E_General_ProcessCycle.LEAK_TEST_HEIGHT_CHECK;
					
				END_IF

E_General_ProcessCycle.LEAK_TEST_HEIGHT_CHECK:

				stLSS.CMD.LSS_CMD.Measurement1						 			:= bProcessedPart[0];
				stLSS.CMD.LSS_CMD.Measurement2						 			:= bProcessedPart[1];
				stLSS.CMD.bExecute												:= TRUE;

				stLeakTesters.CMD.LeakTestersCMD.RunLeakTester1					:= bProcessedPart[0];
				stLeakTesters.CMD.LeakTestersCMD.RunLeakTester2					:= bProcessedPart[1];
				stLeakTesters.CMD.bExecute										:= TRUE;
				
				IF tonExecute.Q THEN
					
					eCycleState													:= E_General_ProcessCycle.WAIT_LEAK_TEST_HEIGHT_CHECK;	
					
				END_IF

E_General_ProcessCycle.WAIT_LEAK_TEST_HEIGHT_CHECK:

				IF stLeakTesters.Status.bDone AND stLSS.Status.bDone THEN
					
					stLeakTesters.CMD.bExecute									:= FALSE;
					stLeakTesters.CMD.LeakTestersCMD.RunLeakTester1				:= FALSE;
					stLeakTesters.CMD.LeakTestersCMD.RunLeakTester2				:= FALSE;
					
					stLSS.CMD.LSS_CMD.Measurement1								:= FALSE;
					stLSS.CMD.LSS_CMD.Measurement2								:= FALSE;
					stLSS.CMD.bExecute											:= FALSE;
					
					stLSS.CMD.bAcknowledge 										:= TRUE;				
					stLeakTesters.CMD.bAcknowledge 								:= TRUE;
					
					eCycleState													:= E_General_ProcessCycle.WAIT_RESULTS;
					
				END_IF
				
				
E_General_ProcessCycle.WAIT_RESULTS:

				IF tonGettingResults.Q THEN
					
					eCycleState													:= E_General_ProcessCycle.RESULTS;
					
				END_IF


E_General_ProcessCycle.RESULTS:

				
					
					IF bProcessedPart[0] THEN
					
						IF stCycleDataNest1.LeakTest_Pass AND stCycleDataNest1.LSS_Pass AND stCycleDataNest1.Camera_Pass THEN	
				
							stCycleDataNest1.bPass								:= TRUE;
							stCycleDataNest1.bFail								:= FALSE;
				
						ELSE stCycleDataNest1.bFail								:= TRUE;
							stCycleDataNest1.bPass								:= FALSE;
				
						END_IF
					
					END_IF
				
					IF bProcessedPart[1] THEN
					
						IF stCycleDataNest2.LeakTest_Pass (*AND stCycleDataNest2.LSS_Pass*) AND stCycleDataNest2.Camera_Pass THEN	
				
							stCycleDataNest2.bPass								:= TRUE;
							stCycleDataNest2.bFail								:= FALSE;
				
						ELSE stCycleDataNest2.bFail								:= TRUE;
							stCycleDataNest2.bPass								:= FALSE;
				
						END_IF
					
					END_IF				
				
				stCycleDataNest1.sTime											:= sSystemTime;
				stCycleDataNest1.sDate											:= sSystemDate;
				stCycleDataNest2.sTime											:= sSystemTime;
				stCycleDataNest2.sDate											:= sSystemDate;
					
				eCycleState														:= E_General_ProcessCycle.WAIT_TO_SAVE_DATA;
									
E_General_ProcessCycle.WAIT_TO_SAVE_DATA:
				
				IF tonExecute.Q THEN
					
					eCycleState													:= E_General_ProcessCycle.SAVE_DATA;	
					
				END_IF

E_General_ProcessCycle.SAVE_DATA:

				IF bProcessedPart[0] THEN
					
					FOR i := 199 TO 0 BY -1 DO
						
						aDataHistoryNest1[i+1] 									:= aDataHistoryNest1[i];
						
					END_FOR
				
				END_IF
				
				IF bProcessedPart[1] THEN
					
					FOR i := 199 TO 0 BY -1 DO
						
						aDataHistoryNest2[i+1] 									:= aDataHistoryNest2[i];
						
					END_FOR
				
				END_IF		
			
				eCycleState														:= E_General_ProcessCycle.SAVE_DATA2;
					
E_General_ProcessCycle.SAVE_DATA2:	
				
				
				c_ACT_SaveData();	
								
				eCycleState														:= E_General_ProcessCycle.CSV_NEST1;
				
				
E_General_ProcessCycle.CSV_NEST1:

				IF bProcessedPart[0] THEN
					
					bWriteNest1													:= TRUE;
					
					IF bCSVDone OR bCSVError THEN
						
						bWriteNest1												:= FALSE;
						bCSVError												:= FALSE;
						
						eCycleState												:= E_General_ProcessCycle.CSV_NEST2;
						
					END_IF
					
				ELSE eCycleState												:= E_General_ProcessCycle.CSV_NEST2;				
					
				END_IF
			
				
E_General_ProcessCycle.CSV_NEST2:

				IF bCSVDone THEN
					
						bWriteNest2												:= FALSE;
						eCycleState												:= E_General_ProcessCycle.VACUUM_CYLINDER_RETRACTION;	
	
				END_IF

				IF bProcessedPart[1] AND  bCSVReady AND NOT bCSVDone AND NOT bCSVError THEN
				
						bWriteNest2												:= TRUE;

				ELSIF NOT bProcessedPart[1] OR bCSVError THEN

						 eCycleState											:= E_General_ProcessCycle.VACUUM_CYLINDER_RETRACTION;
						 bCSVError												:= FALSE;
						 
				END_IF
				
E_General_ProcessCycle.VACUUM_CYLINDER_RETRACTION:

				stVacuumCylinder.CMD.VacuumCylinderCMD.Retract1					:= bProcessedPart[0];
				stVacuumCylinder.CMD.VacuumCylinderCMD.Retract2					:= bProcessedPart[1];
				stVacuumCylinder.CMD.bExecute									:= TRUE;
					
				IF tonExecute.Q THEN
					
					eCycleState													:= E_General_ProcessCycle.WAIT_VACUUM_CYLINDER_RETRACTION;	
					
				END_IF

E_General_ProcessCycle.WAIT_VACUUM_CYLINDER_RETRACTION:

				IF stVacuumCylinder.Status.bDone THEN
					
					stVacuumCylinder.CMD.VacuumCylinderCMD.Extend1				:= FALSE;
					stVacuumCylinder.CMD.VacuumCylinderCMD.Extend2				:= FALSE;
					stVacuumCylinder.CMD.bExecute								:= FALSE;
					stLSS.CMD.bAcknowledge 										:= TRUE;	
					
					eCycleState													:= E_General_ProcessCycle.RELEASE_PART;
					
				END_IF	

E_General_ProcessCycle.RELEASE_PART:	

				stProcessCylinder.CMD.ProcessCylinderCMD.RetractPartHolder1		:= bProcessedPart[0];
				stProcessCylinder.CMD.ProcessCylinderCMD.RetractPartHolder2		:= bProcessedPart[1];
				stProcessCylinder.CMD.bExecute									:= TRUE;
					
				IF tonExecute.Q THEN
					
					eCycleState													:= E_General_ProcessCycle.WAIT_RELEASE_PART;	
					
				END_IF	

E_General_ProcessCycle.WAIT_RELEASE_PART:	

				IF stProcessCylinder.Status.bDone THEN
					
					stProcessCylinder.CMD.ProcessCylinderCMD.RetractPartHolder1	:= FALSE;
					stProcessCylinder.CMD.ProcessCylinderCMD.RetractPartHolder1	:= FALSE;
					stProcessCylinder.CMD.bExecute								:= FALSE;
					stProcessCylinder.CMD.bAcknowledge							:= TRUE;	
					
					eCycleState													:= E_General_ProcessCycle.RETRACT_PROCESS_CYLINDER;
					
				END_IF				
				
E_General_ProcessCycle.RETRACT_PROCESS_CYLINDER:
						
				stProcessCylinder.CMD.ProcessCylinderCMD.RetractCylinder1		:= bProcessedPart[0];
				stProcessCylinder.CMD.ProcessCylinderCMD.RetractCylinder2		:= bProcessedPart[1];	
				stProcessCylinder.CMD.bExecute									:= TRUE;
				
				IF tonExecute.Q THEN
					
					eCycleState													:= E_General_ProcessCycle.WAIT_RETRACT_PROCESS_CYLINDER;	
					
				END_IF

E_General_ProcessCycle.WAIT_RETRACT_PROCESS_CYLINDER:

				IF 	stProcessCylinder.Status.bDone THEN
					
					stProcessCylinder.CMD.ProcessCylinderCMD.RetractCylinder1	:= FALSE;
					stProcessCylinder.CMD.ProcessCylinderCMD.RetractCylinder2	:= FALSE;
					stProcessCylinder.CMD.bExecute								:= FALSE;
					stProcessCylinder.CMD.bAcknowledge							:= TRUE;
					
					IF NOT bEmptyRejectChute THEN

						eCycleState							:= E_General_ProcessCycle.OPEN_PROCESS_DOOR;
					
					ELSE eCycleState							:= E_General_ProcessCycle.REJECT_CHUTE_FULL; 
					
					END_IF
					
				END_IF
	
E_General_ProcessCycle.REJECT_CHUTE_FULL:

				sMachineMessage									:= 'Waiting for Reject chute empty';

				IF NOT bEmptyRejectChute THEN
					
						sMachineMessage							:= '';
						eCycleState								:= E_General_ProcessCycle.OPEN_PROCESS_DOOR;
				
				END_IF	
		
E_General_ProcessCycle.OPEN_PROCESS_DOOR:

				stProcessDoor.CMD.ProcessDoorCMD.OpenDoor						:= TRUE;
				stProcessDoor.CMD.bExecute										:= TRUE;
				
				IF tonExecute.Q THEN
					
					eCycleState													:= E_General_ProcessCycle.WAIT_OPEN_PROCESS_DOOR;	
					
				END_IF

E_General_ProcessCycle.WAIT_OPEN_PROCESS_DOOR:

				IF 	stProcessDoor.Status.bDone THEN
					
					stProcessDoor.CMD.ProcessDoorCMD.OpenDoor					:= FALSE;
					stProcessDoor.CMD.bExecute									:= FALSE;
					stProcessDoor.CMD.bAcknowledge								:= TRUE;
					
					eCycleState													:= E_General_ProcessCycle.PUCK_DEFINITION;
					
				END_IF

E_General_ProcessCycle.PUCK_DEFINITION:
		
				(* Renan Added - Buglist n6 - 08Jul26 *)
				bCycleHasFailure := (bProcessedPart[0] AND stCycleDataNest1.bFail) OR (bProcessedPart[1] AND stCycleDataNest2.bFail);

				bCycleAllProcessedPass := (bProcessedPart[0] OR bProcessedPart[1]) AND ((NOT bProcessedPart[0]) OR stCycleDataNest1.bPass) AND ((NOT bProcessedPart[1]) OR stCycleDataNest2.bPass);
					(*\Renan Added - Buglist n6 - 08Jul26 *)
					
					(* Renan Added 10Jul26 - Puck Locker *)
				IF bPuckLockerEnable AND bCycleAllProcessedPass THEN
					
					GVL_Stations.stPuckLocker.nRequestedRelease := USINT#0;
					
					IF bProcessedPart[0] AND stCycleDataNest1.bPass THEN
						
						GVL_Stations.stPuckLocker.nRequestedRelease := GVL_Stations.stPuckLocker.nRequestedRelease + USINT#1;
						
					END_IF
					
					IF bProcessedPart[1] AND stCycleDataNest2.bPass THEN
						
						GVL_Stations.stPuckLocker.nRequestedRelease := GVL_Stations.stPuckLocker.nRequestedRelease + USINT#1;
							
					END_IF
					
					GVL_Stations.stPuckLocker.bApplyDisposition := TRUE;
					
				END_IF
				
				
				IF bCycleHasFailure THEN //Bugfix 08Jul26
					
					eCycleState								:= E_General_ProcessCycle.WAIT_REJECT_PART;
					
				ELSIF bCycleAllProcessedPass THEN //Bugfix 08Jul26

					eCycleState								:= E_General_ProcessCycle.NEST_CLEARING;
						
				END_IF				
								
E_General_ProcessCycle.WAIT_REJECT_PART:
				
				stCamera.CMD.CameraCMD.ContinuousPartPresent1					:= bProcessedPart[0];
				stCamera.CMD.CameraCMD.ContinuousPartPresent2					:= bProcessedPart[1];
				stCamera.CMD.bExecute											:= TRUE;
					
				ctuRejectPart.CU 												:= rRejectSensor.Q;				

				
				
				IF stCycleDataNest1.bFail AND NOT stCycleDataNest2.bFail THEN
					
					sMachineMessage												:= 'REMOVE PART FROM NEST 1 AND PUT IN REJECT CHUTE';
					
					IF ctuRejectPart.CV > 0 AND NOT bPartPresentNest1 AND (bPartPresentNest2 OR NOT bProcessedPart[1])  THEN
						
						(* Renan Added 10Jul26 - Puck Locker *)
						IF bPuckLockerEnable THEN
							GVL_Stations.stPuckLocker.nRequestedRelease 		:= USINT#1;
							GVL_Stations.stPuckLocker.bApplyDisposition 		:= TRUE;
						END_IF
						(*\Renan Added 10Jul26 - Puck Locker *)
						
						eCycleState												:= E_General_ProcessCycle.NEST_CLEARING;
						
					ELSIF ctuRejectPart.CV > 0 AND (bPartPresentNest1 OR (NOT bPartPresentNest2 AND bProcessedPart[1])) THEN
						
						bRejectPartFault										:= TRUE; 
					
					END_IF
					
					IF NOT bPartPresentNest2 AND bProcessedPart[1] THEN
						
						bRejectPartDialog[0]									:= TRUE;		
						sMachineMessage											:= 'WRONG PART TAKEN';
						
					ELSIF  bPartPresentNest2 THEN
						
						bRejectPartDialog[0]									:= FALSE;
						
					END_IF					
					
				ELSIF NOT stCycleDataNest1.bFail AND stCycleDataNest2.bFail THEN
					
					sMachineMessage												:= 'REMOVE PART FROM NEST 2 AND PUT IN REJECT CHUTE';
					
					IF ctuRejectPart.CV > 0 AND NOT bPartPresentNest2 AND (bPartPresentNest1 OR NOT bProcessedPart[0])  THEN
						
						(* Renan Added 10Jul26 - Puck Locker *)
						IF bPuckLockerEnable THEN
							GVL_Stations.stPuckLocker.nRequestedRelease 		:= USINT#1;
							GVL_Stations.stPuckLocker.bApplyDisposition 		:= TRUE;
						END_IF
						(*\Renan Added 10Jul26 - Puck Locker *)
						
						eCycleState												:= E_General_ProcessCycle.NEST_CLEARING;
						
					ELSIF ctuRejectPart.CV > 0 AND (bPartPresentNest1 OR (NOT bPartPresentNest1 AND bProcessedPart[0])) THEN
						
						bRejectPartFault										:= TRUE; 
					
					END_IF
					
					IF NOT bPartPresentNest1 AND bProcessedPart[0] THEN
						
						bRejectPartDialog[1]									:= TRUE;		
						sMachineMessage											:= 'WRONG PART TAKEN';
						
					ELSIF  bPartPresentNest1 THEN
						
						bRejectPartDialog[1]									:= FALSE;
						
					END_IF
				
